# B&R Automation Studio project NAINV104C00R8L515F00
Automation Studio 4.8.4.50 SP; technology packages: Acp10Arnc0 3.18.2, mapp 1.65.1

## Configuration Inverter_Std

CPU X20CP0483, AutomationRuntime B4.82, Build 4.1.2, Safety 0.0, Vc V4.72.1

### Task classes (Cpu.sw)
```
Cyclic#1 (cycle 10000 us, tolerance 10000 us):
  DInput <- DInput.DInput.prg  // l
  DOutput <- DOutput.DOutput.prg
Cyclic#2 (cycle 20000 us, tolerance 20000 us):
  MotorBrk1 <- MotorBrk.MotorBrk.prg
  Conv <- Conv.Conv.prg
Cyclic#3 (cycle 50000 us, tolerance 50000 us):
  General <- General.General.prg
  UsrFolder <- UsrFolder.UsrFolder.prg
  Time <- Time.Time.prg
  Alarm <- Alarm.Alarm.prg
  RstErr <- RstErr.RstErr.prg
  UsrMgmt <- UsrMgmt.UsrMgmt.prg
  LibVer <- LibVer.LibVer.prg
  PneuNoSenS <- Pneu.PneuNoSenStopper.prg
  PneuNoSenC <- Pneu.PneuNoSenClamp.prg
  Pneu2SenIn <- Pneu.Pneu2SenInShutter.prg
  Pneu2SenOu <- Pneu.Pneu2SenOutShutter.prg
  Pneu2SenI1 <- Pneu.Pneu2SenInClamp1.prg
  Pneu2SenI2 <- Pneu.Pneu2SenInClamp2.prg
  Pneu2SenI3 <- Pneu.Pneu2SenInClamp3.prg
  TLBuz <- TLBuz.TLBuz.prg
  HWInfo <- HWInfo.HWInfo.prg
  ProdRcp <- ProdRcp.ProdRcp.prg
  MpProdRcp <- MpProdRcp.MpProdRcp.prg
  LCS <- LCS.LCS.prg
  LCSMngRcp <- LCS.LCSMngRcp.prg
  LCSLF <- LCS.LCSLF.prg
  Startup <- Startup.Startup.prg
  Machine <- Machine.Machine.prg
  USSMEMA <- SMEMA.USSMEMA.prg
  DSSMEMA <- SMEMA.DSSMEMA.prg
  Hermes <- Hermes.Hermes.prg
  USHermes <- Hermes.USHermes.prg
  DSHermes <- Hermes.DSHermes.prg
  RmtHermes <- Hermes.RmtHermes.prg
  LFLeader <- LF.LFLeader.prg
  LFFollower <- LF.LFFollower.prg
  Follower1 <- LF.Follower1.prg
  AWOpen <- CANOpenServo.AW.AWOpen.prg
  Ops <- Operations.Ops.prg
  OpsInvert <- Operations.OpsInvert.prg
  McParam <- McParam.McParam.prg
  NtParam <- NtParam.NtParam.prg
  UI <- UI.UI.prg
Cyclic#4 (cycle 10000 us, tolerance 10000 us):
  Simu <- Simulation.Simu.prg
  SimuInv <- Simulation.SimuInv.prg
DataObjects: Acp10sys
VcDataObjects: Visu <- UI.Visu.dob
Binaries: vccdt, vccbmp, Visu03, vcfile, arial, vctcal, arialxsr, vcmgr, vccstr, vcbclass, vccbtn, vcgclass, vcdsint, vcnet, vccline, vcshared, vccddbox, arialbd, vccnum, vcpdvnc, vcpdsw, visvc, vccslider, vccbar, vcctext, Visu01, arialbi, vcfntttf, vccovl, vccshape, vcalarm, vcpkat, Visu02, vcrt, udbdef, vccpopup, vcdsloc, vcchspot, TCData, vcpfgen, arsvcreg, Acp10map, acp10cfg, Config, iomap, User, sysconf, ashwac, ashwd, Role, asfw, arconfig, OpcUaMap, vcpfar00, segoeuib, vcctrend
Libraries: standard, astime, asstring, AsCANopen, visapi, FileIO, AsIODiag, AsMem, dvframe, AsOpcUac, sys_lib, AsTCP, runtime, AsIecCon, AsIORTI, MpRecipe, MpCom, Acp10_MC, brsystem, Acp10man, NcGlobal, Acp10par, AsFltGen, MpBase, AsUSB, vcresman, powerlnk, dataobj, asarcfg, NtUSB, NtRecipe, NtUI, NtGeneral, NtHermes
```

### Hardware
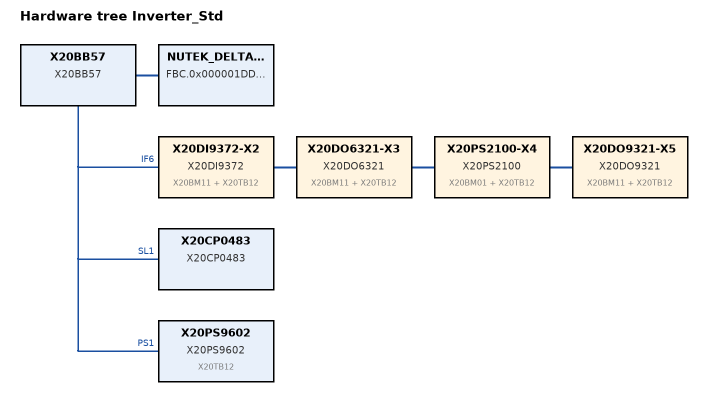
```
NUTEK_DELTA_V101 : FBC.0x000001DD.0x00000001.NUTEK_DELTA_EDS_V101 v1.0 (OrderNumber=NUTEK_DELTA_V101)  [CAN1 -> X20BB57.IF7 (NodeNumber=16)]
X20BB57 : X20BB57 v1.1.1.0
  Connector IF7:
    Baudrate = 1000000
    ActivateCanOpen = 1
    p100c_parametervalue = 1000
    p100d_parametervalue = 3
X20BM01a : X20BM01 v2.1.0.0  [X2X1 -> X20BM11c.X2X2]
X20BM11 : X20BM11 v1.0.0.1  [X2X1 -> X20BB57.IF6]
X20BM11b : X20BM11 v1.0.0.1  [X2X1 -> X20BM01a.X2X2]
X20BM11c : X20BM11 v1.0.0.1  [X2X1 -> X20BM11.X2X2]
X20CP0483 : X20CP0483 v1.2.1.0  [SL -> X20BB57.SL1]
  Connector IF2:
    ActivateDevice = 1
    Mode = Manual
    InternetAddress = 192.168.0.34
    SubnetMask = 255.255.255.0
    InaNodeNumber = 34
    Vnc1
    VncVcObjectName1 = Visu
    VncKeyMappingFile1 = VC\PS2-Keyboard.dis
    VncMaxConnections1 = 3
    VncRefreshRate1 = 100
    ActivateSnmp = 2
  ConfigurationID = NAINV104
  UserPartitionSize = 150
  EnableUsbRemoteInstall = 1
  TimerDeviceType = SWIOTIMER
  Cyclic1Duration = 10000
  Cyclic1Tolerance = 10000
  Cyclic2Duration = 20000
  Cyclic2Tolerance = 20000
  Cyclic3Duration = 50000
  Cyclic3Tolerance = 50000
  Cyclic4Duration = 10000
  Cyclic4Tolerance = 10000
  Cyclic5Duration = 150000
  Cyclic5Tolerance = 150000
  Cyclic6Duration = 500000
  Cyclic6Tolerance = 500000
  Cyclic7Duration = 1000000
  Cyclic7Tolerance = 1000000
  Cyclic8Duration = 10000
  Cyclic8Tolerance = 10000
  FileDevice1
  FileDeviceName1 = F
  FileDevicePath1 = F:
  FileDevice2
  FileDeviceName2 = User
  FileDevicePath2 = F:\User
  FileDevice3
  FileDeviceName3 = Private
  FileDevicePath3 = F:\Private
  FileDevice4
  FileDeviceName4 = CustomerUser
  FileDevicePath4 = F:\User\UserMgmt
  FileDevice5
  FileDeviceName5 = ProdRcp
  FileDevicePath5 = F:\User\ProductRecipe
  FileDevice6
  FileDeviceName6 = MagRcp
  FileDevicePath6 = F:\User\MagazineRecipe
  FileDevice7
  FileDeviceName7 = Alarm
  FileDevicePath7 = F:\User\Alarm
  FileDevice8
  FileDeviceName8 = McParam
  FileDevicePath8 = F:\User\MachineParameter
  FileDevice9
  FileDeviceName9 = NtParam
  FileDevicePath9 = F:\Private\NutekParameter
  FileDevice10
  FileDeviceName10 = LibVer
  FileDevicePath10 = F:\User\LibrariesVersion
  FileDevice11
  FileDeviceName11 = Retain
  FileDevicePath11 = F:\User\Retain
  FileDevice12
  FileDeviceName12 = Log
  FileDevicePath12 = F:\User\Log
  FileDevice13
  FileDeviceName13 = LCS
  FileDevicePath13 = F:\User\LCS
  FileDevice14
  FileDeviceName14 = MpProdRcp
  FileDevicePath14 = F:\User\ProductRecipeXml
  FileDevice15
  FileDeviceName15 = MpNtParam
  FileDevicePath15 = F:\Private\NutekParameterXml
  FtpUser1
  FtpUsername1 = NTAFTP
  FtpUserPassword1 = AX0LBkHXk5z+64iWno3s7Za7qAB1ef/xlwoQUvfPuPs=  // NTA4BH
  FtpUserSalt1 = ulQWWQjW
  FTPAccessRight1 = 0
  FTPdevice1 = ALL
  FtpUser2
  FtpUsername2 = admin
  FtpUserPassword2 = oOnwLF+CCxXL8HlJuADbdqMAHEOaZat9TyrIEGDt79E=  // admin
  FtpUserSalt2 = uTI38Rtv
  FTPAccessRight2 = 0
  FTPMSpath2 = User
  FtpUser3
  FtpUsername3 = LCS
  FtpUserPassword3 = aZ5TTuYKHpukMjerDxdtnomIopt08VfYSbHSRSZ/6LI=  // LCS
  FtpUserSalt3 = ciWQito9
  FTPAccessRight3 = 0
  FTPMSpath3 = User\LCS
  FtpUser4
  FtpUsername4 = user
  FtpUserPassword4 = iZkQD5M0oi0PmKyrQQ/mRhzQwdWVF4GSJtKjbRROesw=  // user
  FtpUserSalt4 = U6prW9t0
  FTPMSpath4 = User\ProductRecipeXml
  ActivateOpcUa = 1
  OpcUaInformationModels_PV_Version = 1
X20DI9372-X2 : X20DI9372 v1.1.0.0  [SS1 -> X20TB12a.SS; SL -> X20BM11.SL1]
X20DO6321-X3 : X20DO6321 v1.1.0.0  [SS1 -> X20TB12c.SS; SL -> X20BM11c.SL1]
X20DO9321-X5 : X20DO9321 v1.1.0.0  [SS1 -> X20TB12f.SS; SL -> X20BM11b.SL1]
X20PS2100-X4 : X20PS2100 v1.2.0.0  [SS1 -> X20TB12d.SS; SL -> X20BM01a.SL1]
X20PS9602 : X20PS9602 v1.0.2.0  [PS -> X20BB57.PS1; SS1 -> X20TB12.SS]
X20TB12 : X20TB12 v1.0.0.0
X20TB12a : X20TB12 v1.0.0.0
X20TB12c : X20TB12 v1.0.0.0
X20TB12d : X20TB12 v1.0.0.0
X20TB12f : X20TB12 v1.0.0.0
```

### IoMap.iom - X20CP0483/IoMap.iom
```iecst
VAR_CONFIG
	::DInput:a_bPhysicalDI[1] AT %IX."X20DI9372-X2".DigitalInput01;
	::DInput:a_bPhysicalDI[2] AT %IX."X20DI9372-X2".DigitalInput02;
	::DInput:a_bPhysicalDI[3] AT %IX."X20DI9372-X2".DigitalInput03;
	::DInput:a_bPhysicalDI[4] AT %IX."X20DI9372-X2".DigitalInput04;
	::DInput:a_bPhysicalDI[5] AT %IX."X20DI9372-X2".DigitalInput05;
	::DInput:a_bPhysicalDI[6] AT %IX."X20DI9372-X2".DigitalInput06;
	::DInput:a_bPhysicalDI[7] AT %IX."X20DI9372-X2".DigitalInput07;
	::DInput:a_bPhysicalDI[8] AT %IX."X20DI9372-X2".DigitalInput08;
	::DInput:a_bPhysicalDI[9] AT %IX."X20DI9372-X2".DigitalInput09;
	::DInput:a_bPhysicalDI[10] AT %IX."X20DI9372-X2".DigitalInput10;
	::DInput:a_bPhysicalDI[11] AT %IX."X20DI9372-X2".DigitalInput11;
	::DInput:a_bPhysicalDI[12] AT %IX."X20DI9372-X2".DigitalInput12;
	::AWOpen:bModuleOK AT %IX."NUTEK_DELTA_V101".ModuleOk;
	::AWOpen:tyParamOutDriver.uiCtrlword_6040 AT %QW."NUTEK_DELTA_V101".Controlword_6040;
	::AWOpen:tyParamInDriver.uiErrCode_603F AT %IW."NUTEK_DELTA_V101".ErrorCode_603F;
	::AWOpen:tyParamInDriver.uiStatword_6041 AT %IW."NUTEK_DELTA_V101".Statusword_6041;
	::AWOpen:tyParamOutDriver.siModOfOpt_6060 AT %QB."NUTEK_DELTA_V101".ModesOfOperation_6060;
	::AWOpen:tyParamInDriver.siModOfOptDisp_6061 AT %IB."NUTEK_DELTA_V101".ModesOfOperationDisplay_6061;
	::AWOpen:tyParamInDriver.diActualPos_6064 AT %ID."NUTEK_DELTA_V101".PositionActualValue_6064;
	::AWOpen:tyParamOutDriver.diTargetPos_607A AT %QD."NUTEK_DELTA_V101".TargetPosition_607A;
	::AWOpen:tyParamOutDriver.udiMoveSpd_6081 AT %QD."NUTEK_DELTA_V101".ProfileVelocity_6081;
	::AWOpen:tyParamOutDriver.siHmMethod_6098 AT %QB."NUTEK_DELTA_V101".HomingMethod_6098;
	::AWOpen:tyParamInDriver.udiDigitalInputs_60FD AT %ID."NUTEK_DELTA_V101".DigitalInputs_60FD;
	::AWOpen:tyParamOutDriver.diJogVel_60FF AT %QD."NUTEK_DELTA_V101".TargetVelocity_60FF;
	::DOutput:a_bPhysicalDO[1] AT %QX."X20DO6321-X3".DigitalOutput01;
	::DOutput:a_bPhysicalDO[2] AT %QX."X20DO6321-X3".DigitalOutput02;
	::DOutput:a_bPhysicalDO[3] AT %QX."X20DO6321-X3".DigitalOutput03;
	::DOutput:a_bPhysicalDO[4] AT %QX."X20DO6321-X3".DigitalOutput04;
	::DOutput:a_bPhysicalDO[5] AT %QX."X20DO6321-X3".DigitalOutput05;
	::DOutput:a_bPhysicalDO[6] AT %QX."X20DO6321-X3".DigitalOutput06;
	::DOutput:a_bPhysicalDO[7] AT %QX."X20DO9321".DigitalOutput01;
	::DOutput:a_bPhysicalDO[8] AT %QX."X20DO9321".DigitalOutput02;
	::DOutput:a_bPhysicalDO[9] AT %QX."X20DO9321".DigitalOutput03;
	::DOutput:a_bPhysicalDO[10] AT %QX."X20DO9321".DigitalOutput04;
	::DOutput:a_bPhysicalDO[11] AT %QX."X20DO9321".DigitalOutput05;
	::DOutput:a_bPhysicalDO[12] AT %QX."X20DO9321".DigitalOutput06;
	::DOutput:a_bPhysicalDO[13] AT %QX."X20DO9321".DigitalOutput07;
	::DOutput:a_bPhysicalDO[14] AT %QX."X20DO9321".DigitalOutput08;
	::DOutput:a_bPhysicalDO[15] AT %QX."X20DO9321".DigitalOutput09;
	::DOutput:a_bPhysicalDO[16] AT %QX."X20DO9321".DigitalOutput10;
	::DOutput:a_bPhysicalDO[17] AT %QX."X20DO9321".DigitalOutput11;
	::DOutput:a_bPhysicalDO[18] AT %QX."X20DO9321".DigitalOutput12;
	::DOutput:a_bPhysicalDO[7] AT %QX."X20DO9321-X5".DigitalOutput01;
	::DOutput:a_bPhysicalDO[8] AT %QX."X20DO9321-X5".DigitalOutput02;
	::DOutput:a_bPhysicalDO[9] AT %QX."X20DO9321-X5".DigitalOutput03;
	::DOutput:a_bPhysicalDO[10] AT %QX."X20DO9321-X5".DigitalOutput04;
	::DOutput:a_bPhysicalDO[11] AT %QX."X20DO9321-X5".DigitalOutput05;
	::DOutput:a_bPhysicalDO[12] AT %QX."X20DO9321-X5".DigitalOutput06;
	::DOutput:a_bPhysicalDO[13] AT %QX."X20DO9321-X5".DigitalOutput07;
	::DOutput:a_bPhysicalDO[14] AT %QX."X20DO9321-X5".DigitalOutput08;
	::DOutput:a_bPhysicalDO[15] AT %QX."X20DO9321-X5".DigitalOutput09;
	::DOutput:a_bPhysicalDO[16] AT %QX."X20DO9321-X5".DigitalOutput10;
	::DOutput:a_bPhysicalDO[17] AT %QX."X20DO9321-X5".DigitalOutput11;
	::DOutput:a_bPhysicalDO[18] AT %QX."X20DO9321-X5".DigitalOutput12;
END_VAR
```

## Configuration Inverter_Std_Estun

CPU X20CP0483, AutomationRuntime B4.82, Build 4.1.2, Vc V4.72.1

### Task classes (Cpu.sw)
```
Cyclic#1 (cycle 10000 us, tolerance 10000 us):
  DInput <- DInput.DInput.prg  // l
  DOutput <- DOutput.DOutput.prg
Cyclic#2 (cycle 20000 us, tolerance 20000 us):
  Conv <- Conv.Conv.prg
Cyclic#3 (cycle 50000 us, tolerance 50000 us):
  General <- General.General.prg
  UsrFolder <- UsrFolder.UsrFolder.prg
  Time <- Time.Time.prg
  Alarm <- Alarm.Alarm.prg
  RstErr <- RstErr.RstErr.prg
  UsrMgmt <- UsrMgmt.UsrMgmt.prg
  LibVer <- LibVer.LibVer.prg
  PneuNoSenS <- Pneu.PneuNoSenStopper.prg
  PneuNoSenC <- Pneu.PneuNoSenClamp.prg
  Pneu2SenIn <- Pneu.Pneu2SenInShutter.prg
  Pneu2SenOu <- Pneu.Pneu2SenOutShutter.prg
  Pneu2SenI1 <- Pneu.Pneu2SenInClamp1.prg
  Pneu2SenI2 <- Pneu.Pneu2SenInClamp2.prg
  Pneu2SenI3 <- Pneu.Pneu2SenInClamp3.prg
  TLBuz <- TLBuz.TLBuz.prg
  HWInfo <- HWInfo.HWInfo.prg
  ProdRcp <- ProdRcp.ProdRcp.prg
  MpProdRcp <- MpProdRcp.MpProdRcp.prg
  LCS <- LCS.LCS.prg
  LCSMngRcp <- LCS.LCSMngRcp.prg
  LCSLF <- LCS.LCSLF.prg
  Startup <- Startup.Startup.prg
  Machine <- Machine.Machine.prg
  MotorBrk1 <- MotorBrk.MotorBrk.prg
  USSMEMA <- SMEMA.USSMEMA.prg
  DSSMEMA <- SMEMA.DSSMEMA.prg
  Hermes <- Hermes.Hermes.prg
  USHermes <- Hermes.USHermes.prg
  DSHermes <- Hermes.DSHermes.prg
  RmtHermes <- Hermes.RmtHermes.prg
  LFLeader <- LF.LFLeader.prg
  LFFollower <- LF.LFFollower.prg
  Follower1 <- LF.Follower1.prg
  AWOpen <- CANOpenServo.AW.AWOpen.prg
  Ops <- Operations.Ops.prg
  OpsInvert <- Operations.OpsInvert.prg
  McParam <- McParam.McParam.prg
  NtParam <- NtParam.NtParam.prg
  UI <- UI.UI.prg
Cyclic#4 (cycle 10000 us, tolerance 10000 us):
  Simu <- Simulation.Simu.prg
  SimuInv <- Simulation.SimuInv.prg
DataObjects: Acp10sys
VcDataObjects: Visu <- UI.Visu.dob
Binaries: vccdt, vccbmp, Visu03, vcfile, arial, vctcal, vcmgr, vccstr, vcbclass, vccbtn, vcgclass, vcdsint, vcnet, vccline, vcshared, vccddbox, arialbd, vccnum, vcpdvnc, vcpdsw, visvc, vccslider, vccbar, vcctext, Visu01, arialbi, vcfntttf, vccovl, vccshape, vcalarm, vcpkat, Visu02, vcrt, udbdef, vccpopup, vcdsloc, vcchspot, TCData, arialxsr, vcpfgen, Acp10map, acp10cfg, Config, iomap, User, sysconf, ashwac, ashwd, Role, asfw, arconfig, vcpfar00, OpcUaMap, arsvcreg, segoeuib, vcctrend
Libraries: standard, astime, asstring, AsCANopen, visapi, FileIO, AsIODiag, AsMem, dvframe, AsOpcUac, sys_lib, AsTCP, runtime, AsIecCon, AsIORTI, MpRecipe, MpCom, Acp10_MC, brsystem, Acp10man, NcGlobal, Acp10par, AsFltGen, MpBase, AsUSB, NtMem, vcresman, powerlnk, NtBuffer, NtOvenInfo, NtRS232, NtStepper, NtFileIO, NtLogFile, NtTLBuz, NtMotion, NtPneu, NtConv, NtTCP, NtMessage, NtSMEMA, NtOPCUA, NtVersion, dataobj, asarcfg, NtLF, NtRecipe, NtUI, NtGeneral, NtHermes
```

### Hardware
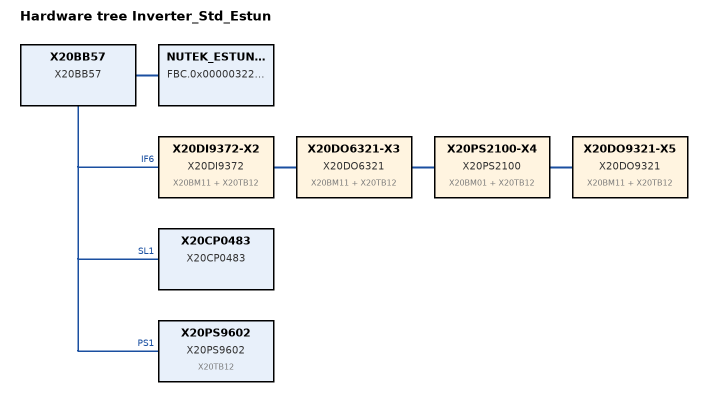
```
NUTEK_ESTUN_PronetPlus_V106 : FBC.0x00000322.0x00001000.NUTEK_ESTUN_PronetPlus_EDS_V106 v1.06.1 (OrderNumber=NUTEK_ESTUN_PronetPlus_V106)  [CAN1 -> X20BB57.IF7 (NodeNumber=16)]
X20BB57 : X20BB57 v1.1.1.0
  Connector IF7:
    Baudrate = 1000000
    ActivateCanOpen = 1
    p100c_parametervalue = 1000
    p100d_parametervalue = 3
X20BM01 : X20BM01 v2.1.0.0  [X2X1 -> X20BM11e.X2X2]
X20BM11 : X20BM11 v1.0.0.1  [X2X1 -> X20BB57.IF6]
X20BM11c : X20BM11 v1.0.0.1  [X2X1 -> X20BM01.X2X2]
X20BM11e : X20BM11 v1.0.0.1  [X2X1 -> X20BM11.X2X2]
X20CP0483 : X20CP0483 v1.2.1.0  [SL -> X20BB57.SL1]
  Connector IF2:
    ActivateDevice = 1
    Mode = Manual
    InternetAddress = 192.168.0.16
    SubnetMask = 255.255.255.0
    InaNodeNumber = 6
    Vnc1
    VncVcObjectName1 = Visu
    VncKeyMappingFile1 = VC\PS2-Keyboard.dis
    VncMaxConnections1 = 3
    VncRefreshRate1 = 100
    ActivateSnmp = 2
  ConfigurationID = NAINV104
  UserPartitionSize = 150
  EnableUsbRemoteInstall = 1
  TimerDeviceType = SWIOTIMER
  Cyclic1Duration = 10000
  Cyclic1Tolerance = 10000
  Cyclic2Duration = 20000
  Cyclic2Tolerance = 20000
  Cyclic3Duration = 50000
  Cyclic3Tolerance = 50000
  Cyclic4Duration = 10000
  Cyclic4Tolerance = 10000
  Cyclic5Duration = 150000
  Cyclic5Tolerance = 150000
  Cyclic6Duration = 500000
  Cyclic6Tolerance = 500000
  Cyclic7Duration = 1000000
  Cyclic7Tolerance = 1000000
  Cyclic8Duration = 10000
  Cyclic8Tolerance = 10000
  FileDevice1
  FileDeviceName1 = F
  FileDevicePath1 = F:
  FileDevice2
  FileDeviceName2 = User
  FileDevicePath2 = F:\User
  FileDevice3
  FileDeviceName3 = Private
  FileDevicePath3 = F:\Private
  FileDevice4
  FileDeviceName4 = CustomerUser
  FileDevicePath4 = F:\User\UserMgmt
  FileDevice5
  FileDeviceName5 = ProdRcp
  FileDevicePath5 = F:\User\ProductRecipe
  FileDevice6
  FileDeviceName6 = MagRcp
  FileDevicePath6 = F:\User\MagazineRecipe
  FileDevice7
  FileDeviceName7 = Alarm
  FileDevicePath7 = F:\User\Alarm
  FileDevice8
  FileDeviceName8 = McParam
  FileDevicePath8 = F:\User\MachineParameter
  FileDevice9
  FileDeviceName9 = NtParam
  FileDevicePath9 = F:\Private\NutekParameter
  FileDevice10
  FileDeviceName10 = LibVer
  FileDevicePath10 = F:\User\LibrariesVersion
  FileDevice11
  FileDeviceName11 = Retain
  FileDevicePath11 = F:\User\Retain
  FileDevice12
  FileDeviceName12 = Log
  FileDevicePath12 = F:\User\Log
  FileDevice13
  FileDeviceName13 = LCS
  FileDevicePath13 = F:\User\LCS
  FileDevice14
  FileDeviceName14 = MpProdRcp
  FileDevicePath14 = F:\User\ProductRecipeXml
  FileDevice15
  FileDeviceName15 = MpNtParam
  FileDevicePath15 = F:\Private\NutekParameterXml
  FtpUser1
  FtpUsername1 = NTAFTP
  FtpUserPassword1 = AX0LBkHXk5z+64iWno3s7Za7qAB1ef/xlwoQUvfPuPs=  // NTA4BH
  FtpUserSalt1 = ulQWWQjW
  FTPAccessRight1 = 0
  FTPdevice1 = ALL
  FtpUser2
  FtpUsername2 = admin
  FtpUserPassword2 = oOnwLF+CCxXL8HlJuADbdqMAHEOaZat9TyrIEGDt79E=  // admin
  FtpUserSalt2 = uTI38Rtv
  FTPAccessRight2 = 0
  FTPMSpath2 = User
  FtpUser3
  FtpUsername3 = LCS
  FtpUserPassword3 = aZ5TTuYKHpukMjerDxdtnomIopt08VfYSbHSRSZ/6LI=  // LCS
  FtpUserSalt3 = ciWQito9
  FTPAccessRight3 = 0
  FTPMSpath3 = User\LCS
  FtpUser4
  FtpUsername4 = user
  FtpUserPassword4 = JD0vxhfsk4AIsU4iEBcqNCfGv1QGBPStLuK1j+bofBk=  // user
  FtpUserSalt4 = BS0DW2Vk
  FTPMSpath4 = User\ProductRecipeXml
  ActivateOpcUa = 1
  OpcUaInformationModels_PV_Version = 1
X20DI9372-X2 : X20DI9372 v1.1.0.0  [SS1 -> X20TB12a.SS; SL -> X20BM11.SL1]
X20DO6321-X3 : X20DO6321 v1.1.0.0  [SS1 -> X20TB12e.SS; SL -> X20BM11e.SL1]
X20DO9321-X5 : X20DO9321 v1.1.0.0  [SS1 -> X20TB12c.SS; SL -> X20BM11c.SL1]
X20PS2100-X4 : X20PS2100 v1.2.0.0  [SS1 -> X20TB12f.SS; SL -> X20BM01.SL1]
X20PS9602 : X20PS9602 v1.0.2.0  [PS -> X20BB57.PS1; SS1 -> X20TB12.SS]
X20TB12 : X20TB12 v1.0.0.0
X20TB12a : X20TB12 v1.0.0.0
X20TB12c : X20TB12 v1.0.0.0
X20TB12e : X20TB12 v1.0.0.0
X20TB12f : X20TB12 v1.0.0.0
```

### IoMap.iom - X20CP0483/IoMap.iom
```iecst
VAR_CONFIG
	::DOutput:a_bPhysicalDO[7] AT %QX."X20DO9321-X5".DigitalOutput01;
	::DOutput:a_bPhysicalDO[8] AT %QX."X20DO9321-X5".DigitalOutput02;
	::DOutput:a_bPhysicalDO[9] AT %QX."X20DO9321-X5".DigitalOutput03;
	::DOutput:a_bPhysicalDO[10] AT %QX."X20DO9321-X5".DigitalOutput04;
	::DOutput:a_bPhysicalDO[11] AT %QX."X20DO9321-X5".DigitalOutput05;
	::DOutput:a_bPhysicalDO[12] AT %QX."X20DO9321-X5".DigitalOutput06;
	::DOutput:a_bPhysicalDO[13] AT %QX."X20DO9321-X5".DigitalOutput07;
	::DOutput:a_bPhysicalDO[14] AT %QX."X20DO9321-X5".DigitalOutput08;
	::DOutput:a_bPhysicalDO[15] AT %QX."X20DO9321-X5".DigitalOutput09;
	::DOutput:a_bPhysicalDO[16] AT %QX."X20DO9321-X5".DigitalOutput10;
	::DOutput:a_bPhysicalDO[17] AT %QX."X20DO9321-X5".DigitalOutput11;
	::DOutput:a_bPhysicalDO[18] AT %QX."X20DO9321-X5".DigitalOutput12;
	::DInput:a_bPhysicalDI[1] AT %IX."X20DI9372-X2".DigitalInput01;
	::DInput:a_bPhysicalDI[2] AT %IX."X20DI9372-X2".DigitalInput02;
	::DInput:a_bPhysicalDI[3] AT %IX."X20DI9372-X2".DigitalInput03;
	::DInput:a_bPhysicalDI[4] AT %IX."X20DI9372-X2".DigitalInput04;
	::DInput:a_bPhysicalDI[5] AT %IX."X20DI9372-X2".DigitalInput05;
	::DInput:a_bPhysicalDI[6] AT %IX."X20DI9372-X2".DigitalInput06;
	::DInput:a_bPhysicalDI[7] AT %IX."X20DI9372-X2".DigitalInput07;
	::DInput:a_bPhysicalDI[8] AT %IX."X20DI9372-X2".DigitalInput08;
	::DInput:a_bPhysicalDI[9] AT %IX."X20DI9372-X2".DigitalInput09;
	::DInput:a_bPhysicalDI[10] AT %IX."X20DI9372-X2".DigitalInput10;
	::DInput:a_bPhysicalDI[11] AT %IX."X20DI9372-X2".DigitalInput11;
	::DInput:a_bPhysicalDI[12] AT %IX."X20DI9372-X2".DigitalInput12;
	::DOutput:a_bPhysicalDO[1] AT %QX."X20DO6321-X3".DigitalOutput01;
	::DOutput:a_bPhysicalDO[2] AT %QX."X20DO6321-X3".DigitalOutput02;
	::DOutput:a_bPhysicalDO[3] AT %QX."X20DO6321-X3".DigitalOutput03;
	::DOutput:a_bPhysicalDO[4] AT %QX."X20DO6321-X3".DigitalOutput04;
	::DOutput:a_bPhysicalDO[5] AT %QX."X20DO6321-X3".DigitalOutput05;
	::DOutput:a_bPhysicalDO[6] AT %QX."X20DO6321-X3".DigitalOutput06;
	::AWOpen:bModuleOK AT %IX."NUTEK_ESTUN_PronetPlus_V106".ModuleOk;
	::AWOpen:tyParamInDriver.uiErrCode_603F AT %IW."NUTEK_ESTUN_PronetPlus_V106".Error_code_603F;
	::AWOpen:tyParamOutDriver.uiCtrlword_6040 AT %QW."NUTEK_ESTUN_PronetPlus_V106".Controlword_6040;
	::AWOpen:tyParamInDriver.uiStatword_6041 AT %IW."NUTEK_ESTUN_PronetPlus_V106".Statusword_6041;
	::AWOpen:tyParamOutDriver.siModOfOpt_6060 AT %QB."NUTEK_ESTUN_PronetPlus_V106".Modes_of_operation_6060;
	::AWOpen:tyParamInDriver.siModOfOptDisp_6061 AT %IB."NUTEK_ESTUN_PronetPlus_V106".Modes_of_operation_display_6061;
	::AWOpen:tyParamInDriver.diActualPos_6064 AT %ID."NUTEK_ESTUN_PronetPlus_V106".Position_actual_value_6064;
	::AWOpen:tyParamOutDriver.diTargetPos_607A AT %QD."NUTEK_ESTUN_PronetPlus_V106".Target_position_607A;
	::AWOpen:tyParamOutDriver.udiMoveSpd_6081 AT %QD."NUTEK_ESTUN_PronetPlus_V106".Profile_velocity_6081;
	::AWOpen:tyParamOutDriver.siHmMethod_6098 AT %QB."NUTEK_ESTUN_PronetPlus_V106".Homing_method_6098;
	::AWOpen:tyParamInDriver.udiDigitalInputs_60FD AT %ID."NUTEK_ESTUN_PronetPlus_V106".Digital_intputs_60FD;
	::AWOpen:tyParamOutDriver.diJogVel_60FF AT %QD."NUTEK_ESTUN_PronetPlus_V106".Target_velocity_60FF;
END_VAR
```

## Configuration Inverter_XClamp_WShutter_

### Hardware
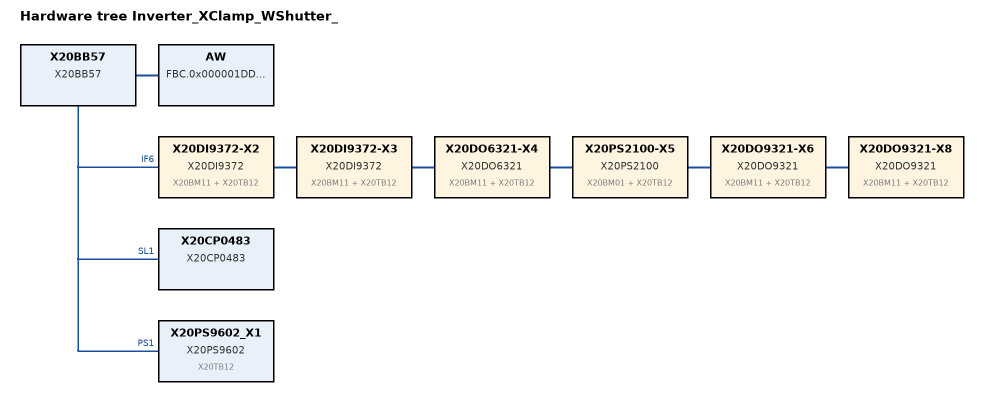
```
AW : FBC.0x000001DD.0x00000001.NUTEK_DELTA_EDS_V101 v1.0 (OrderNumber=NUTEK_DELTA_V101)  [CAN1 -> X20BB57.IF7 (NodeNumber=16)]
  Supervision = on
X20BB57 : X20BB57 v1.1.1.0
  Connector IF7:
    Baudrate = 1000000
    ActivateCanOpen = 1
    p100c_parametervalue = 1000
    p100d_parametervalue = 3
X20BM01 : X20BM01 v2.1.0.0  [X2X1 -> X20BM11a.X2X2]
X20BM11 : X20BM11 v1.0.0.1  [X2X1 -> X20BB57.IF6]
X20BM11a : X20BM11 v1.0.0.1  [X2X1 -> X20BM11e.X2X2]
X20BM11b : X20BM11 v1.0.0.1  [X2X1 -> X20BM01.X2X2]
X20BM11e : X20BM11 v1.0.0.1  [X2X1 -> X20BM11.X2X2]
X20BM11g : X20BM11 v1.0.0.1  [X2X1 -> X20BM11b.X2X2]
X20CP0483 : X20CP0483 v1.2.1.0  [SL -> X20BB57.SL1]
  Connector IF2:
    ActivateDevice = 1
    Mode = Manual
    InternetAddress = 192.168.0.30
    SubnetMask = 255.255.255.0
    InaNodeNumber = 42
    Vnc1
    VncVcObjectName1 = Visu
    VncKeyMappingFile1 = VC\PS2-Keyboard.dis
    VncMaxConnections1 = 3
    VncRefreshRate1 = 100
    ActivateSnmp = 2
  ConfigurationID = NAINV104
  UserPartitionSize = 150
  EnableUsbRemoteInstall = 1
  TimerDeviceType = SWIOTIMER
  Cyclic1Duration = 10000
  Cyclic1Tolerance = 10000
  Cyclic2Duration = 20000
  Cyclic2Tolerance = 20000
  Cyclic3Duration = 50000
  Cyclic3Tolerance = 50000
  Cyclic4Duration = 10000
  Cyclic4Tolerance = 10000
  Cyclic5Duration = 150000
  Cyclic5Tolerance = 150000
  Cyclic6Duration = 500000
  Cyclic6Tolerance = 500000
  Cyclic7Duration = 1000000
  Cyclic7Tolerance = 1000000
  Cyclic8Duration = 10000
  Cyclic8Tolerance = 10000
  FileDevice1
  FileDeviceName1 = F
  FileDevicePath1 = F:
  FileDevice2
  FileDeviceName2 = User
  FileDevicePath2 = F:\User
  FileDevice3
  FileDeviceName3 = Private
  FileDevicePath3 = F:\Private
  FileDevice4
  FileDeviceName4 = CustomerUser
  FileDevicePath4 = F:\User\UserMgmt
  FileDevice5
  FileDeviceName5 = ProdRcp
  FileDevicePath5 = F:\User\ProductRecipe
  FileDevice6
  FileDeviceName6 = MagRcp
  FileDevicePath6 = F:\User\MagazineRecipe
  FileDevice7
  FileDeviceName7 = Alarm
  FileDevicePath7 = F:\User\Alarm
  FileDevice8
  FileDeviceName8 = McParam
  FileDevicePath8 = F:\User\MachineParameter
  FileDevice9
  FileDeviceName9 = NtParam
  FileDevicePath9 = F:\Private\NutekParameter
  FileDevice10
  FileDeviceName10 = LibVer
  FileDevicePath10 = F:\User\LibrariesVersion
  FileDevice11
  FileDeviceName11 = Retain
  FileDevicePath11 = F:\User\Retain
  FileDevice12
  FileDeviceName12 = Log
  FileDevicePath12 = F:\User\Log
  FileDevice13
  FileDeviceName13 = LCS
  FileDevicePath13 = F:\User\LCS
  FileDevice14
  FileDeviceName14 = MpProdRcp
  FileDevicePath14 = F:\User\ProductRecipeXml
  FileDevice15
  FileDeviceName15 = MpNtParam
  FileDevicePath15 = F:\Private\NutekParameterXml
  FtpUser1
  FtpUsername1 = NTAFTP
  FtpUserPassword1 = AX0LBkHXk5z+64iWno3s7Za7qAB1ef/xlwoQUvfPuPs=  // NTA4BH
  FtpUserSalt1 = ulQWWQjW
  FTPAccessRight1 = 0
  FTPdevice1 = ALL
  FtpUser2
  FtpUsername2 = admin
  FtpUserPassword2 = oOnwLF+CCxXL8HlJuADbdqMAHEOaZat9TyrIEGDt79E=  // admin
  FtpUserSalt2 = uTI38Rtv
  FTPAccessRight2 = 0
  FTPMSpath2 = User
  FtpUser3
  FtpUsername3 = LCS
  FtpUserPassword3 = aZ5TTuYKHpukMjerDxdtnomIopt08VfYSbHSRSZ/6LI=  // LCS
  FtpUserSalt3 = ciWQito9
  FTPAccessRight3 = 0
  FTPMSpath3 = User\LCS
  FtpUser4
  FtpUsername4 = user
  FtpUserPassword4 = ZSNVrCTF84rK225EpwbOTF9hgjmxleDX5xeb+GcCkC0=
  FtpUserSalt4 = jV67T8tr
  FTPMSpath4 = User\ProductRecipeXml
  ActivateOpcUa = 1
  OpcUa_ConversationSecurityPolicy_EnableBasic256Rsa256 = 0
  OpcUaInformationModels_PV_Version = 1
X20DI9372-X2 : X20DI9372 v1.1.0.0  [SS1 -> X20TB12a.SS; SL -> X20BM11.SL1]
X20DI9372-X3 : X20DI9372 v1.1.0.0  [SS1 -> X20TB12g.SS; SL -> X20BM11e.SL1]
X20DO6321-X4 : X20DO6321 v1.1.0.0  [SS1 -> X20TB12b.SS; SL -> X20BM11a.SL1]
X20DO9321-X6 : X20DO9321 v1.1.0.0  [SS1 -> X20TB12c.SS; SL -> X20BM11b.SL1]
X20DO9321-X8 : X20DO9321 v1.1.0.0  [SS1 -> X20TB12i.SS; SL -> X20BM11g.SL1]
X20PS2100-X5 : X20PS2100 v1.2.0.0  [SS1 -> X20TB12f.SS; SL -> X20BM01.SL1]
X20PS9602_X1 : X20PS9602 v1.0.2.0  [PS -> X20BB57.PS1; SS1 -> X20TB12.SS]
X20TB12 : X20TB12 v1.0.0.0
X20TB12a : X20TB12 v1.0.0.0
X20TB12b : X20TB12 v1.0.0.0
X20TB12c : X20TB12 v1.0.0.0
X20TB12f : X20TB12 v1.0.0.0
X20TB12g : X20TB12 v1.0.0.0
X20TB12i : X20TB12 v1.0.0.0
```

### IoMap.iom - X20CP0483/IoMap.iom
```iecst
VAR_CONFIG
	::DInput:a_bPhysicalDI[1] AT %IX."X20DI9372-X2".DigitalInput01; (*safety relay*)
	::DInput:a_bPhysicalDI[2] AT %IX."X20DI9372-X2".DigitalInput02; (*e-stop*)
	::DInput:a_bPhysicalDI[3] AT %IX."X20DI9372-X2".DigitalInput03; (*cover swicth*)
	::DInput:a_bPhysicalDI[4] AT %IX."X20DI9372-X2".DigitalInput04; (*uba*)
	::DInput:a_bPhysicalDI[5] AT %IX."X20DI9372-X2".DigitalInput05; (*dsb*)
	::DInput:a_bPhysicalDI[6] AT %IX."X20DI9372-X2".DigitalInput06;
	::DInput:a_bPhysicalDI[7] AT %IX."X20DI9372-X2".DigitalInput07; (*inlet sen*)
	::DInput:a_bPhysicalDI[8] AT %IX."X20DI9372-X2".DigitalInput08; (*outlet sen*)
	::DInput:a_bPhysicalDI[9] AT %IX."X20DI9372-X2".DigitalInput09; (*hm inv*)
	::DInput:a_bPhysicalDI[10] AT %IX."X20DI9372-X2".DigitalInput10; (*rmt inv*)
	::DInput:a_bPhysicalDI[11] AT %IX."X20DI9372-X2".DigitalInput11; (*stp blk*)
	::DInput:a_bPhysicalDI[12] AT %IX."X20DI9372-X2".DigitalInput12; (*stp unblk*)
	::DOutput:a_bPhysicalDO[1] AT %QX."X20DO6321-X4".DigitalOutput01; (*safety relay reset*)
	::DOutput:a_bPhysicalDO[2] AT %QX."X20DO6321-X4".DigitalOutput02; (*TL G*)
	::DOutput:a_bPhysicalDO[3] AT %QX."X20DO6321-X4".DigitalOutput03; (*TL A*)
	::DOutput:a_bPhysicalDO[4] AT %QX."X20DO6321-X4".DigitalOutput04; (*TL R*)
	::DOutput:a_bPhysicalDO[5] AT %QX."X20DO6321-X4".DigitalOutput05; (*Buz*)
	::DOutput:a_bPhysicalDO[6] AT %QX."X20DO6321-X4".DigitalOutput06;
	::DOutput:a_bPhysicalDO[7] AT %QX."X20DO9321-X6".DigitalOutput01;
	::DOutput:a_bPhysicalDO[8] AT %QX."X20DO9321-X6".DigitalOutput02; (*USB*)
	::DOutput:a_bPhysicalDO[9] AT %QX."X20DO9321-X6".DigitalOutput03; (*DBA*)
	::DOutput:a_bPhysicalDO[10] AT %QX."X20DO9321-X6".DigitalOutput04;
	::DOutput:a_bPhysicalDO[11] AT %QX."X20DO9321-X6".DigitalOutput05; (*Conv Mtr CW*)
	::DOutput:a_bPhysicalDO[12] AT %QX."X20DO9321-X6".DigitalOutput06; (*Conv Mtr CWW*)
	::DOutput:a_bPhysicalDO[13] AT %QX."X20DO9321-X6".DigitalOutput07; (*Stpr ublk *)
	::DOutput:a_bPhysicalDO[14] AT %QX."X20DO9321-X6".DigitalOutput08; (*Stpr blk*)
	::DOutput:a_bPhysicalDO[15] AT %QX."X20DO9321-X6".DigitalOutput09; (*inv hm*)
	::DOutput:a_bPhysicalDO[16] AT %QX."X20DO9321-X6".DigitalOutput10; (*inv rmt*)
	::DOutput:a_bPhysicalDO[17] AT %QX."X20DO9321-X6".DigitalOutput11; (*inv brake*)
	::DOutput:a_bPhysicalDO[18] AT %QX."X20DO9321-X6".DigitalOutput12;
	::AWOpen:bModuleOK AT %IX."AW".ModuleOk;
	::AWOpen:tyParamOutDriver.uiCtrlword_6040 AT %QW."AW".Controlword_6040;
	::AWOpen:tyParamInDriver.uiStatword_6041 AT %IW."AW".Statusword_6041;
	::DInput:a_bPhysicalDI[13] AT %IX."X20DI6372".DigitalInput01;
	::DInput:a_bPhysicalDI[14] AT %IX."X20DI6372".DigitalInput02;
	::DInput:a_bPhysicalDI[15] AT %IX."X20DI6372".DigitalInput03;
	::DInput:a_bPhysicalDI[16] AT %IX."X20DI6372".DigitalInput04;
	::DInput:a_bPhysicalDI[17] AT %IX."X20DI6372".DigitalInput05;
	::DInput:a_bPhysicalDI[18] AT %IX."X20DI6372".DigitalInput06;
	::AWOpen:tyParamOutDriver.siModOfOpt_6060 AT %QB."AW".ModesOfOperation_6060;
	::AWOpen:tyParamInDriver.siModOfOptDisp_6061 AT %IB."AW".ModesOfOperationDisplay_6061;
	::AWOpen:tyParamInDriver.diActualPos_6064 AT %ID."AW".PositionActualValue_6064;
	::AWOpen:tyParamOutDriver.diTargetPos_607A AT %QD."AW".TargetPosition_607A;
	::AWOpen:tyParamOutDriver.udiMoveSpd_6081 AT %QD."AW".ProfileVelocity_6081;
	::AWOpen:tyParamOutDriver.siHmMethod_6098 AT %QB."AW".HomingMethod_6098;
	::AWOpen:tyParamInDriver.udiDigitalInputs_60FD AT %ID."AW".DigitalInputs_60FD;
	::AWOpen:tyParamOutDriver.diJogVel_60FF AT %QD."AW".TargetVelocity_60FF;
	::DInput:a_bPhysicalDI[13] AT %IX."X20DI9372-X3".DigitalInput01; (*inlet shut close reed*)
	::DInput:a_bPhysicalDI[14] AT %IX."X20DI9372-X3".DigitalInput02; (*inlet shut open reed*)
	::DInput:a_bPhysicalDI[15] AT %IX."X20DI9372-X3".DigitalInput03; (*oulet close reed*)
	::DInput:a_bPhysicalDI[16] AT %IX."X20DI9372-X3".DigitalInput04; (*outlet open reed*)
	::DInput:a_bPhysicalDI[17] AT %IX."X20DI9372-X3".DigitalInput05;
	::DInput:a_bPhysicalDI[18] AT %IX."X20DI9372-X3".DigitalInput06;
	::DInput:a_bPhysicalDI[19] AT %IX."X20DI9372-X3".DigitalInput07;
	::DInput:a_bPhysicalDI[20] AT %IX."X20DI9372-X3".DigitalInput08;
	::DInput:a_bPhysicalDI[21] AT %IX."X20DI9372-X3".DigitalInput09;
	::DInput:a_bPhysicalDI[22] AT %IX."X20DI9372-X3".DigitalInput10;
	::DInput:a_bPhysicalDI[23] AT %IX."X20DI9372-X3".DigitalInput11;
	::DInput:a_bPhysicalDI[24] AT %IX."X20DI9372-X3".DigitalInput12;
	::DOutput:a_bPhysicalDO[19] AT %QX."X20DO9321-X8".DigitalOutput01; (*inlet shut close*)
	::DOutput:a_bPhysicalDO[20] AT %QX."X20DO9321-X8".DigitalOutput02; (*inlet shut open*)
	::DOutput:a_bPhysicalDO[21] AT %QX."X20DO9321-X8".DigitalOutput03; (*outlet shut close*)
	::DOutput:a_bPhysicalDO[22] AT %QX."X20DO9321-X8".DigitalOutput04; (*outlet shut open*)
	::DOutput:a_bPhysicalDO[23] AT %QX."X20DO9321-X8".DigitalOutput05;
	::AWOpen:tyParamInDriver.uiErrCode_603F AT %IW."AW".ErrorCode_603F;
	::DOutput:a_bPhysicalDO[24] AT %QX."X20DO9321-X8".DigitalOutput06;
	::DOutput:a_bPhysicalDO[25] AT %QX."X20DO9321-X8".DigitalOutput07;
	::DOutput:a_bPhysicalDO[26] AT %QX."X20DO9321-X8".DigitalOutput08;
	::DOutput:a_bPhysicalDO[27] AT %QX."X20DO9321-X8".DigitalOutput09;
	::DOutput:a_bPhysicalDO[28] AT %QX."X20DO9321-X8".DigitalOutput10;
	::DOutput:a_bPhysicalDO[29] AT %QX."X20DO9321-X8".DigitalOutput11;
	::DOutput:a_bPhysicalDO[30] AT %QX."X20DO9321-X8".DigitalOutput12;
END_VAR
```

## Configuration Inverter_XStd_WClamp

CPU X20CP0483, AutomationRuntime B4.34, Build 4.1.2, Vc V4.33.0

### Task classes (Cpu.sw)
```
Cyclic#1 (cycle 10000 us, tolerance 10000 us):
  DInput <- DInput.DInput.prg
  DOutput <- DOutput.DOutput.prg
Cyclic#2 (cycle 20000 us, tolerance 20000 us):
  Conv <- Conv.Conv.prg
Cyclic#3 (cycle 50000 us, tolerance 50000 us):
  General <- General.General.prg
  UsrFolder <- UsrFolder.UsrFolder.prg
  Time <- Time.Time.prg
  Alarm <- Alarm.Alarm.prg
  RstErr <- RstErr.RstErr.prg
  UsrMgmt <- UsrMgmt.UsrMgmt.prg
  LibVer <- LibVer.LibVer.prg
  PneuNoSenS <- Pneu.PneuNoSenStopper.prg
  PneuNoSenC <- Pneu.PneuNoSenClamp.prg
  Pneu2SenIn <- Pneu.Pneu2SenInShutter.prg
  Pneu2SenOu <- Pneu.Pneu2SenOutShutter.prg
  Pneu2SenI1 <- Pneu.Pneu2SenInClamp1.prg
  Pneu2SenI2 <- Pneu.Pneu2SenInClamp2.prg
  Pneu2SenI3 <- Pneu.Pneu2SenInClamp3.prg
  TLBuz <- TLBuz.TLBuz.prg
  HWInfo <- HWInfo.HWInfo.prg
  LCS <- LCS.LCS.prg
  LCSMngRcp <- LCS.LCSMngRcp.prg
  Startup <- Startup.Startup.prg
  LCSLF <- LCS.LCSLF.prg
  Machine <- Machine.Machine.prg
  MotorBrk1 <- MotorBrk.MotorBrk.prg
  USSMEMA <- SMEMA.USSMEMA.prg
  DSSMEMA <- SMEMA.DSSMEMA.prg
  Hermes <- Hermes.Hermes.prg
  USHermes <- Hermes.USHermes.prg
  DSHermes <- Hermes.DSHermes.prg
  RmtHermes <- Hermes.RmtHermes.prg
  LFLeader <- LF.LFLeader.prg
  LFFollower <- LF.LFFollower.prg
  Follower1 <- LF.Follower1.prg
  AWOpen <- CANOpenServo.AW.AWOpen.prg
  Ops <- Operations.Ops.prg
  OpsInvert <- Operations.OpsInvert.prg
  McParam <- McParam.McParam.prg
  NtParam <- NtParam.NtParam.prg
  UI <- UI.UI.prg
  MpProdRcp <- MpProdRcp.MpProdRcp.prg
  ProdRcp <- ProdRcp.ProdRcp.prg
Cyclic#4 (cycle 10000 us, tolerance 10000 us):
  Simu <- Simulation.Simu.prg
  SimuInv <- Simulation.SimuInv.prg
DataObjects: Acp10sys
VcDataObjects: Visu <- UI.Visu.dob
Binaries: vccdt, vccbmp, Visu03, vcfile, arial, vctcal, arialxsr, vcmgr, vccstr, vcbclass, vccbtn, vcgclass, vcdsint, vcnet, vccline, vcshared, vccddbox, arialbd, vccnum, vcpdvnc, vcpdsw, visvc, vccslider, vccbar, vcctext, Visu01, arialbi, vcfntttf, vccovl, vccshape, vcalarm, vcpkat, Visu02, vcrt, udbdef, vccpopup, vcdsloc, vcchspot, TCData, arsvcreg, vcpfgen, arconfig, asfw, Role, ashwd, ashwac, sysconf, User, OpcUaMap, iomap, Config, acp10cfg, Acp10map, vcpfar00, segoeuib, vcctrend
Libraries: standard, astime, asstring, AsCANopen, visapi, FileIO, AsIODiag, AsMem, dvframe, AsOpcUac, sys_lib, AsTCP, runtime, AsIecCon, AsIORTI, MpRecipe, MpCom, Acp10_MC, brsystem, Acp10man, NcGlobal, Acp10par, AsFltGen, MpBase, AsRfbExt, AsUSB, vcresman, dataobj, powerlnk, asarcfg, NtRecipe, NtUI, NtGeneral, NtHermes
```

### Hardware
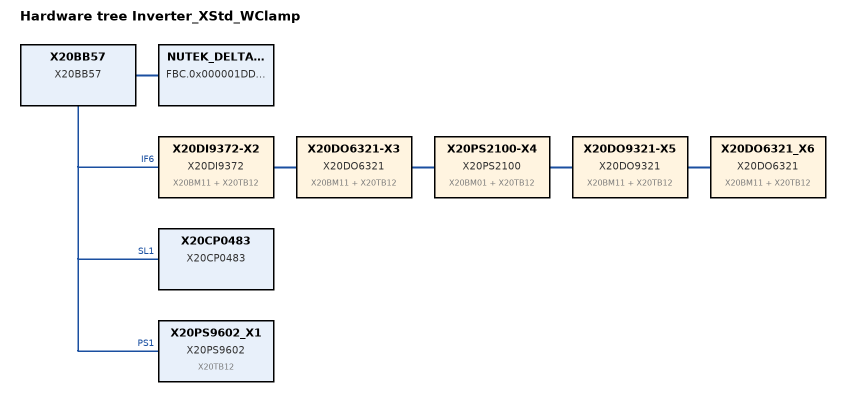
```
NUTEK_DELTA_V101 : FBC.0x000001DD.0x00000001.NUTEK_DELTA_EDS_V101 v1.0 (OrderNumber=NUTEK_DELTA_V101)  [CAN1 -> X20BB57.IF7 (NodeNumber=16)]
  Supervision = on
X20BB57 : X20BB57 v1.1.1.0
  Connector IF7:
    Baudrate = 1000000
    ActivateCanOpen = 1
    p100c_parametervalue = 1000
    p100d_parametervalue = 3
X20BM01 : X20BM01 v2.1.0.0  [X2X1 -> X20BM11a.X2X2]
X20BM11 : X20BM11 v1.0.0.1  [X2X1 -> X20BB57.IF6]
X20BM11a : X20BM11 v1.0.0.1  [X2X1 -> X20BM11.X2X2]
X20BM11b : X20BM11 v1.0.0.1  [X2X1 -> X20BM01.X2X2]
X20BM11d : X20BM11 v1.0.0.1  [X2X1 -> X20BM11b.X2X2]
X20CP0483 : X20CP0483 v1.2.1.0  [SL -> X20BB57.SL1]
  Connector IF2:
    ActivateDevice = 1
    Mode = Manual
    InternetAddress = 192.168.0.6
    SubnetMask = 255.255.255.0
    InaNodeNumber = 6
    Vnc1
    VncVcObjectName1 = Visu
    VncKeyMappingFile1 = VC\PS2-Keyboard.dis
    VncMaxConnections1 = 3
    VncRefreshRate1 = 100
  ConfigurationID = NAINV104
  UserPartitionSize = 150
  EnableUsbRemoteInstall = 1
  TimerDeviceType = SWIOTIMER
  Cyclic1Duration = 10000
  Cyclic1Tolerance = 10000
  Cyclic2Duration = 20000
  Cyclic2Tolerance = 20000
  Cyclic3Duration = 50000
  Cyclic3Tolerance = 50000
  Cyclic4Duration = 10000
  Cyclic4Tolerance = 10000
  Cyclic5Duration = 150000
  Cyclic5Tolerance = 150000
  Cyclic6Duration = 500000
  Cyclic6Tolerance = 500000
  Cyclic7Duration = 1000000
  Cyclic7Tolerance = 1000000
  Cyclic8Duration = 10000
  Cyclic8Tolerance = 10000
  FileDevice1
  FileDeviceName1 = F
  FileDevicePath1 = F:
  FileDevice2
  FileDeviceName2 = User
  FileDevicePath2 = F:\User
  FileDevice3
  FileDeviceName3 = Private
  FileDevicePath3 = F:\Private
  FileDevice4
  FileDeviceName4 = CustomerUser
  FileDevicePath4 = F:\User\UserMgmt
  FileDevice5
  FileDeviceName5 = ProdRcp
  FileDevicePath5 = F:\User\ProductRecipe
  FileDevice6
  FileDeviceName6 = MagRcp
  FileDevicePath6 = F:\User\MagazineRecipe
  FileDevice7
  FileDeviceName7 = Alarm
  FileDevicePath7 = F:\User\Alarm
  FileDevice8
  FileDeviceName8 = McParam
  FileDevicePath8 = F:\User\MachineParameter
  FileDevice9
  FileDeviceName9 = NtParam
  FileDevicePath9 = F:\Private\NutekParameter
  FileDevice10
  FileDeviceName10 = LibVer
  FileDevicePath10 = F:\User\LibrariesVersion
  FileDevice11
  FileDeviceName11 = Retain
  FileDevicePath11 = F:\User\Retain
  FileDevice12
  FileDeviceName12 = Log
  FileDevicePath12 = F:\User\Log
  FileDevice13
  FileDeviceName13 = LCS
  FileDevicePath13 = F:\User\LCS
  FileDevice14
  FileDeviceName14 = MpProdRcp
  FileDevicePath14 = F:\User\ProductRecipeXml
  FileDevice15
  FileDeviceName15 = MpNtParam
  FileDevicePath15 = F:\Private\NutekParameterXml
  FtpUser1
  FtpUsername1 = NTAFTP
  FtpUserPassword1 = AX0LBkHXk5z+64iWno3s7Za7qAB1ef/xlwoQUvfPuPs=  // NTA4BH
  FtpUserSalt1 = ulQWWQjW
  FTPAccessRight1 = 0
  FTPdevice1 = ALL
  FtpUser2
  FtpUsername2 = admin
  FtpUserPassword2 = oOnwLF+CCxXL8HlJuADbdqMAHEOaZat9TyrIEGDt79E=  // admin
  FtpUserSalt2 = uTI38Rtv
  FTPAccessRight2 = 0
  FTPMSpath2 = User
  FtpUser3
  FtpUsername3 = LCS
  FtpUserPassword3 = aZ5TTuYKHpukMjerDxdtnomIopt08VfYSbHSRSZ/6LI=  // LCS
  FtpUserSalt3 = ciWQito9
  FTPAccessRight3 = 0
  FTPMSpath3 = User\LCS
  FtpUser4
  FtpUsername4 = user
  FtpUserPassword4 = iCt/72nJS6I3I2E3ul1RgkpC9BzXhJ9PtEYmUm0QYyA=  // user
  FtpUserSalt4 = 7DfIs+80
  FTPMSpath4 = User\ProductRecipeXml
  ActivateOpcUa = 1
X20DI9372-X2 : X20DI9372 v1.1.0.0  [SS1 -> X20TB12a.SS; SL -> X20BM11.SL1]
X20DO6321-X3 : X20DO6321 v1.1.0.0  [SS1 -> X20TB12b.SS; SL -> X20BM11a.SL1]
X20DO6321_X6 : X20DO6321 v1.1.0.0  [SS1 -> X20TB12e.SS; SL -> X20BM11d.SL1]
X20DO9321-X5 : X20DO9321 v1.1.0.0  [SS1 -> X20TB12c.SS; SL -> X20BM11b.SL1]
X20PS2100-X4 : X20PS2100 v1.2.0.0  [SS1 -> X20TB12f.SS; SL -> X20BM01.SL1]
X20PS9602_X1 : X20PS9602 v1.0.2.0  [PS -> X20BB57.PS1; SS1 -> X20TB12.SS]
X20TB12 : X20TB12 v1.0.0.0
X20TB12a : X20TB12 v1.0.0.0
X20TB12b : X20TB12 v1.0.0.0
X20TB12c : X20TB12 v1.0.0.0
X20TB12e : X20TB12 v1.0.0.0
X20TB12f : X20TB12 v1.0.0.0
```

### IoMap.iom - X20CP0483/IoMap.iom
```iecst
VAR_CONFIG
	::DInput:a_bPhysicalDI[1] AT %IX."X20DI9372-X2".DigitalInput01;
	::DInput:a_bPhysicalDI[2] AT %IX."X20DI9372-X2".DigitalInput02;
	::DInput:a_bPhysicalDI[3] AT %IX."X20DI9372-X2".DigitalInput03;
	::DInput:a_bPhysicalDI[4] AT %IX."X20DI9372-X2".DigitalInput04;
	::DInput:a_bPhysicalDI[5] AT %IX."X20DI9372-X2".DigitalInput05;
	::DInput:a_bPhysicalDI[6] AT %IX."X20DI9372-X2".DigitalInput06;
	::DInput:a_bPhysicalDI[7] AT %IX."X20DI9372-X2".DigitalInput07;
	::DInput:a_bPhysicalDI[8] AT %IX."X20DI9372-X2".DigitalInput08;
	::DInput:a_bPhysicalDI[9] AT %IX."X20DI9372-X2".DigitalInput09;
	::DInput:a_bPhysicalDI[10] AT %IX."X20DI9372-X2".DigitalInput10;
	::DInput:a_bPhysicalDI[11] AT %IX."X20DI9372-X2".DigitalInput11;
	::DInput:a_bPhysicalDI[12] AT %IX."X20DI9372-X2".DigitalInput12;
	::DOutput:a_bPhysicalDO[1] AT %QX."X20DO6321-X3".DigitalOutput01;
	::DOutput:a_bPhysicalDO[2] AT %QX."X20DO6321-X3".DigitalOutput02;
	::DOutput:a_bPhysicalDO[3] AT %QX."X20DO6321-X3".DigitalOutput03;
	::DOutput:a_bPhysicalDO[4] AT %QX."X20DO6321-X3".DigitalOutput04;
	::DOutput:a_bPhysicalDO[5] AT %QX."X20DO6321-X3".DigitalOutput05;
	::DOutput:a_bPhysicalDO[6] AT %QX."X20DO6321-X3".DigitalOutput06;
	::DOutput:a_bPhysicalDO[7] AT %QX."X20DO9321-X5".DigitalOutput01;
	::DOutput:a_bPhysicalDO[8] AT %QX."X20DO9321-X5".DigitalOutput02;
	::DOutput:a_bPhysicalDO[9] AT %QX."X20DO9321-X5".DigitalOutput03;
	::DOutput:a_bPhysicalDO[10] AT %QX."X20DO9321-X5".DigitalOutput04;
	::DOutput:a_bPhysicalDO[11] AT %QX."X20DO9321-X5".DigitalOutput05;
	::DOutput:a_bPhysicalDO[12] AT %QX."X20DO9321-X5".DigitalOutput06;
	::DOutput:a_bPhysicalDO[13] AT %QX."X20DO9321-X5".DigitalOutput07;
	::DOutput:a_bPhysicalDO[14] AT %QX."X20DO9321-X5".DigitalOutput08;
	::DOutput:a_bPhysicalDO[15] AT %QX."X20DO9321-X5".DigitalOutput09;
	::DOutput:a_bPhysicalDO[16] AT %QX."X20DO9321-X5".DigitalOutput10;
	::DOutput:a_bPhysicalDO[17] AT %QX."X20DO9321-X5".DigitalOutput11;
	::DOutput:a_bPhysicalDO[18] AT %QX."X20DO9321-X5".DigitalOutput12;
	::AWOpen:bModuleOK AT %IX."NUTEK_DELTA_V101".ModuleOk;
	::AWOpen:tyParamOutDriver.uiCtrlword_6040 AT %QW."NUTEK_DELTA_V101".Controlword_6040;
	::AWOpen:tyParamInDriver.uiStatword_6041 AT %IW."NUTEK_DELTA_V101".Statusword_6041;
	::DInput:a_bPhysicalDI[13] AT %IX."X20DI6372".DigitalInput01;
	::DInput:a_bPhysicalDI[14] AT %IX."X20DI6372".DigitalInput02;
	::DInput:a_bPhysicalDI[15] AT %IX."X20DI6372".DigitalInput03;
	::DInput:a_bPhysicalDI[16] AT %IX."X20DI6372".DigitalInput04;
	::DInput:a_bPhysicalDI[17] AT %IX."X20DI6372".DigitalInput05;
	::DInput:a_bPhysicalDI[18] AT %IX."X20DI6372".DigitalInput06;
	::DOutput:a_bPhysicalDO[19] AT %QX."X20DO6321_X6".DigitalOutput01;
	::DOutput:a_bPhysicalDO[20] AT %QX."X20DO6321_X6".DigitalOutput02;
	::DOutput:a_bPhysicalDO[21] AT %QX."X20DO6321_X6".DigitalOutput03;
	::DOutput:a_bPhysicalDO[22] AT %QX."X20DO6321_X6".DigitalOutput04;
	::DOutput:a_bPhysicalDO[23] AT %QX."X20DO6321_X6".DigitalOutput05;
	::DOutput:a_bPhysicalDO[24] AT %QX."X20DO6321_X6".DigitalOutput06;
END_VAR
```

## Configuration Inverter_XStd_WOutShutter_

### Hardware
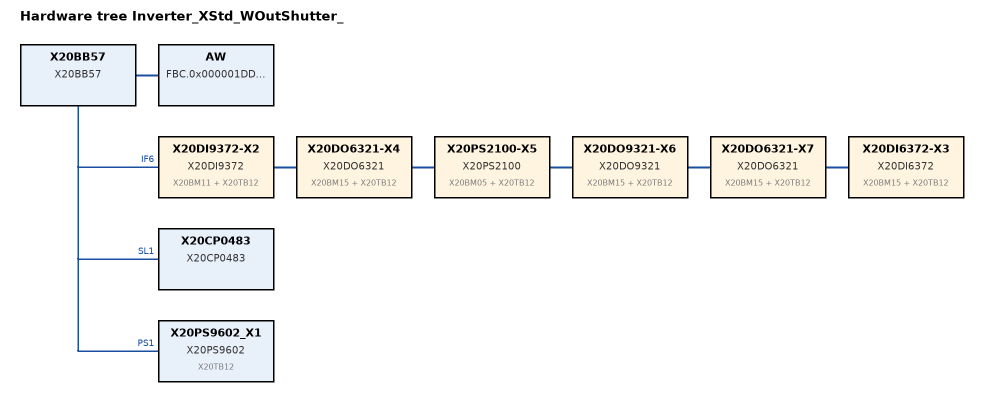
```
AW : FBC.0x000001DD.0x00000001.NUTEK_DELTA_EDS_V101 v1.0 (OrderNumber=NUTEK_DELTA_V101)  [CAN1 -> X20BB57.IF7 (NodeNumber=16)]
  Supervision = on
X20BB57 : X20BB57 v1.1.1.0
  Connector IF7:
    Baudrate = 1000000
    ActivateCanOpen = 1
    p100c_parametervalue = 1000
    p100d_parametervalue = 3
X20BM05 : X20BM05 v1.0.0.3  [X2X1 -> X20BM15b.X2X2 (NodeNumber=4)]
X20BM11 : X20BM11 v1.0.0.1  [X2X1 -> X20BB57.IF6]
X20BM15 : X20BM15 v1.0.1.0  [X2X1 -> X20BM15a.X2X2 (NodeNumber=6)]
X20BM15a : X20BM15 v1.0.1.0  [X2X1 -> X20BM05.X2X2 (NodeNumber=5)]
X20BM15b : X20BM15 v1.0.1.0  [X2X1 -> X20BM11.X2X2 (NodeNumber=3)]
X20BM15c : X20BM15 v1.0.1.0  [X2X1 -> X20BM15.X2X2 (NodeNumber=2)]
X20CP0483 : X20CP0483 v1.2.1.0  [SL -> X20BB57.SL1]
  Connector IF2:
    ActivateDevice = 1
    Mode = Manual
    InternetAddress = 192.168.0.40
    SubnetMask = 255.255.255.0
    InaNodeNumber = 40
    Vnc1
    VncVcObjectName1 = Visu
    VncKeyMappingFile1 = VC\PS2-Keyboard.dis
    VncMaxConnections1 = 3
    VncRefreshRate1 = 100
    ActivateSnmp = 2
  ConfigurationID = NAINV104
  UserPartitionSize = 150
  EnableUsbRemoteInstall = 1
  TimerDeviceType = SWIOTIMER
  Cyclic1Duration = 10000
  Cyclic1Tolerance = 10000
  Cyclic2Duration = 20000
  Cyclic2Tolerance = 20000
  Cyclic3Duration = 50000
  Cyclic3Tolerance = 50000
  Cyclic4Duration = 10000
  Cyclic4Tolerance = 10000
  Cyclic5Duration = 150000
  Cyclic5Tolerance = 150000
  Cyclic6Duration = 500000
  Cyclic6Tolerance = 500000
  Cyclic7Duration = 1000000
  Cyclic7Tolerance = 1000000
  Cyclic8Duration = 10000
  Cyclic8Tolerance = 10000
  FileDevice1
  FileDeviceName1 = F
  FileDevicePath1 = F:
  FileDevice2
  FileDeviceName2 = User
  FileDevicePath2 = F:\User
  FileDevice3
  FileDeviceName3 = Private
  FileDevicePath3 = F:\Private
  FileDevice4
  FileDeviceName4 = CustomerUser
  FileDevicePath4 = F:\User\UserMgmt
  FileDevice5
  FileDeviceName5 = ProdRcp
  FileDevicePath5 = F:\User\ProductRecipe
  FileDevice6
  FileDeviceName6 = MagRcp
  FileDevicePath6 = F:\User\MagazineRecipe
  FileDevice7
  FileDeviceName7 = Alarm
  FileDevicePath7 = F:\User\Alarm
  FileDevice8
  FileDeviceName8 = McParam
  FileDevicePath8 = F:\User\MachineParameter
  FileDevice9
  FileDeviceName9 = NtParam
  FileDevicePath9 = F:\Private\NutekParameter
  FileDevice10
  FileDeviceName10 = LibVer
  FileDevicePath10 = F:\User\LibrariesVersion
  FileDevice11
  FileDeviceName11 = Retain
  FileDevicePath11 = F:\User\Retain
  FileDevice12
  FileDeviceName12 = Log
  FileDevicePath12 = F:\User\Log
  FileDevice13
  FileDeviceName13 = LCS
  FileDevicePath13 = F:\User\LCS
  FileDevice14
  FileDeviceName14 = MpProdRcp
  FileDevicePath14 = F:\User\ProductRecipeXml
  FileDevice15
  FileDeviceName15 = MpNtParam
  FileDevicePath15 = F:\Private\NutekParameterXml
  FtpUser1
  FtpUsername1 = NTAFTP
  FtpUserPassword1 = AX0LBkHXk5z+64iWno3s7Za7qAB1ef/xlwoQUvfPuPs=  // NTA4BH
  FtpUserSalt1 = ulQWWQjW
  FTPAccessRight1 = 0
  FTPdevice1 = ALL
  FtpUser2
  FtpUsername2 = admin
  FtpUserPassword2 = oOnwLF+CCxXL8HlJuADbdqMAHEOaZat9TyrIEGDt79E=  // admin
  FtpUserSalt2 = uTI38Rtv
  FTPAccessRight2 = 0
  FTPMSpath2 = User
  FtpUser3
  FtpUsername3 = LCS
  FtpUserPassword3 = aZ5TTuYKHpukMjerDxdtnomIopt08VfYSbHSRSZ/6LI=  // LCS
  FtpUserSalt3 = ciWQito9
  FTPAccessRight3 = 0
  FTPMSpath3 = User\LCS
  FtpUser4
  FtpUsername4 = user
  FtpUserPassword4 = ZSNVrCTF84rK225EpwbOTF9hgjmxleDX5xeb+GcCkC0=
  FtpUserSalt4 = jV67T8tr
  FTPMSpath4 = User\ProductRecipeXml
  ActivateOpcUa = 1
  OpcUa_ConversationSecurityPolicy_EnableBasic256Rsa256 = 0
  OpcUaInformationModels_PV_Version = 1
X20DI6372-X3 : X20DI6372 v1.1.0.0  [SS1 -> X20TB12d.SS; SL -> X20BM15c.SL1]
X20DI9372-X2 : X20DI9372 v1.1.0.0  [SS1 -> X20TB12a.SS; SL -> X20BM11.SL1]
X20DO6321-X4 : X20DO6321 v1.1.0.0  [SS1 -> X20TB12b.SS; SL -> X20BM15b.SL1]
X20DO6321-X7 : X20DO6321 v1.1.0.0  [SS1 -> X20TB12i.SS; SL -> X20BM15.SL1]
X20DO9321-X6 : X20DO9321 v1.1.0.0  [SS1 -> X20TB12c.SS; SL -> X20BM15a.SL1]
X20PS2100-X5 : X20PS2100 v1.2.0.0  [SS1 -> X20TB12f.SS; SL -> X20BM05.SL1]
X20PS9602_X1 : X20PS9602 v1.0.2.0  [PS -> X20BB57.PS1; SS1 -> X20TB12.SS]
X20TB12 : X20TB12 v1.0.0.0
X20TB12a : X20TB12 v1.0.0.0
X20TB12b : X20TB12 v1.0.0.0
X20TB12c : X20TB12 v1.0.0.0
X20TB12d : X20TB12 v1.0.0.0
X20TB12f : X20TB12 v1.0.0.0
X20TB12i : X20TB12 v1.0.0.0
```

### IoMap.iom - X20CP0483/IoMap.iom
```iecst
VAR_CONFIG
	::DInput:a_bPhysicalDI[1] AT %IX."X20DI9372-X2".DigitalInput01;
	::DInput:a_bPhysicalDI[2] AT %IX."X20DI9372-X2".DigitalInput02;
	::DInput:a_bPhysicalDI[3] AT %IX."X20DI9372-X2".DigitalInput03;
	::DInput:a_bPhysicalDI[4] AT %IX."X20DI9372-X2".DigitalInput04;
	::DInput:a_bPhysicalDI[5] AT %IX."X20DI9372-X2".DigitalInput05;
	::DInput:a_bPhysicalDI[6] AT %IX."X20DI9372-X2".DigitalInput06;
	::DInput:a_bPhysicalDI[7] AT %IX."X20DI9372-X2".DigitalInput07;
	::DInput:a_bPhysicalDI[8] AT %IX."X20DI9372-X2".DigitalInput08;
	::DInput:a_bPhysicalDI[9] AT %IX."X20DI9372-X2".DigitalInput09;
	::DInput:a_bPhysicalDI[10] AT %IX."X20DI9372-X2".DigitalInput10;
	::DInput:a_bPhysicalDI[11] AT %IX."X20DI9372-X2".DigitalInput11;
	::DInput:a_bPhysicalDI[12] AT %IX."X20DI9372-X2".DigitalInput12;
	::DOutput:a_bPhysicalDO[1] AT %QX."X20DO6321-X4".DigitalOutput01;
	::DOutput:a_bPhysicalDO[2] AT %QX."X20DO6321-X4".DigitalOutput02;
	::DOutput:a_bPhysicalDO[3] AT %QX."X20DO6321-X4".DigitalOutput03;
	::DOutput:a_bPhysicalDO[4] AT %QX."X20DO6321-X4".DigitalOutput04;
	::DOutput:a_bPhysicalDO[5] AT %QX."X20DO6321-X4".DigitalOutput05;
	::DOutput:a_bPhysicalDO[6] AT %QX."X20DO6321-X4".DigitalOutput06;
	::DOutput:a_bPhysicalDO[7] AT %QX."X20DO9321-X6".DigitalOutput01;
	::DOutput:a_bPhysicalDO[8] AT %QX."X20DO9321-X6".DigitalOutput02;
	::DOutput:a_bPhysicalDO[9] AT %QX."X20DO9321-X6".DigitalOutput03;
	::DOutput:a_bPhysicalDO[10] AT %QX."X20DO9321-X6".DigitalOutput04;
	::DOutput:a_bPhysicalDO[11] AT %QX."X20DO9321-X6".DigitalOutput05;
	::DOutput:a_bPhysicalDO[12] AT %QX."X20DO9321-X6".DigitalOutput06;
	::DOutput:a_bPhysicalDO[13] AT %QX."X20DO9321-X6".DigitalOutput07;
	::DOutput:a_bPhysicalDO[14] AT %QX."X20DO9321-X6".DigitalOutput08;
	::DOutput:a_bPhysicalDO[15] AT %QX."X20DO9321-X6".DigitalOutput09;
	::DOutput:a_bPhysicalDO[16] AT %QX."X20DO9321-X6".DigitalOutput10;
	::DOutput:a_bPhysicalDO[17] AT %QX."X20DO9321-X6".DigitalOutput11;
	::DOutput:a_bPhysicalDO[18] AT %QX."X20DO9321-X6".DigitalOutput12;
	::AWOpen:bModuleOK AT %IX."AW".ModuleOk;
	::AWOpen:tyParamOutDriver.uiCtrlword_6040 AT %QW."AW".Controlword_6040;
	::AWOpen:tyParamInDriver.uiStatword_6041 AT %IW."AW".Statusword_6041;
	::AWOpen:tyParamOutDriver.siModOfOpt_6060 AT %QB."AW".ModesOfOperation_6060;
	::AWOpen:tyParamInDriver.siModOfOptDisp_6061 AT %IB."AW".ModesOfOperationDisplay_6061;
	::AWOpen:tyParamInDriver.diActualPos_6064 AT %ID."AW".PositionActualValue_6064;
	::AWOpen:tyParamOutDriver.diTargetPos_607A AT %QD."AW".TargetPosition_607A;
	::AWOpen:tyParamOutDriver.udiMoveSpd_6081 AT %QD."AW".ProfileVelocity_6081;
	::AWOpen:tyParamOutDriver.siHmMethod_6098 AT %QB."AW".HomingMethod_6098;
	::AWOpen:tyParamInDriver.udiDigitalInputs_60FD AT %ID."AW".DigitalInputs_60FD;
	::AWOpen:tyParamOutDriver.diJogVel_60FF AT %QD."AW".TargetVelocity_60FF;
	::DOutput:a_bPhysicalDO[19] AT %QX."X20DO6321-X7".DigitalOutput01;
	::DOutput:a_bPhysicalDO[20] AT %QX."X20DO6321-X7".DigitalOutput02;
	::DOutput:a_bPhysicalDO[21] AT %QX."X20DO6321-X7".DigitalOutput03;
	::DOutput:a_bPhysicalDO[22] AT %QX."X20DO6321-X7".DigitalOutput04;
	::DOutput:a_bPhysicalDO[23] AT %QX."X20DO6321-X7".DigitalOutput05;
	::DOutput:a_bPhysicalDO[24] AT %QX."X20DO6321-X7".DigitalOutput06;
	::AWOpen:tyParamInDriver.uiErrCode_603F AT %IW."AW".ErrorCode_603F;
	::DInput:a_bPhysicalDI[13] AT %IX."X20DI6372-X3".DigitalInput01;
	::DInput:a_bPhysicalDI[14] AT %IX."X20DI6372-X3".DigitalInput02;
	::DInput:a_bPhysicalDI[15] AT %IX."X20DI6372-X3".DigitalInput03;
	::DInput:a_bPhysicalDI[16] AT %IX."X20DI6372-X3".DigitalInput04;
	::DInput:a_bPhysicalDI[17] AT %IX."X20DI6372-X3".DigitalInput05;
	::DInput:a_bPhysicalDI[18] AT %IX."X20DI6372-X3".DigitalInput06;
END_VAR
```

## Configuration Inverter_XStd_WShutter

CPU X20CP0483, AutomationRuntime B4.82, Build 4.1.2, Vc V4.72.1

### Task classes (Cpu.sw)
```
Cyclic#1 (cycle 10000 us, tolerance 10000 us):
  DInput <- DInput.DInput.prg
  DOutput <- DOutput.DOutput.prg
Cyclic#2 (cycle 20000 us, tolerance 20000 us):
  Conv <- Conv.Conv.prg
Cyclic#3 (cycle 50000 us, tolerance 50000 us):
  General <- General.General.prg
  UsrFolder <- UsrFolder.UsrFolder.prg
  Time <- Time.Time.prg
  Alarm <- Alarm.Alarm.prg
  RstErr <- RstErr.RstErr.prg
  UsrMgmt <- UsrMgmt.UsrMgmt.prg
  LibVer <- LibVer.LibVer.prg
  PneuNoSenS <- Pneu.PneuNoSenStopper.prg
  PneuNoSenC <- Pneu.PneuNoSenClamp.prg
  Pneu2SenIn <- Pneu.Pneu2SenInShutter.prg
  Pneu2SenOu <- Pneu.Pneu2SenOutShutter.prg
  Pneu2SenI1 <- Pneu.Pneu2SenInClamp1.prg
  Pneu2SenI2 <- Pneu.Pneu2SenInClamp2.prg
  Pneu2SenI3 <- Pneu.Pneu2SenInClamp3.prg
  TLBuz <- TLBuz.TLBuz.prg
  HWInfo <- HWInfo.HWInfo.prg
  LCS <- LCS.LCS.prg
  LCSMngRcp <- LCS.LCSMngRcp.prg
  Startup <- Startup.Startup.prg
  LCSLF <- LCS.LCSLF.prg
  Machine <- Machine.Machine.prg
  MotorBrk1 <- MotorBrk.MotorBrk.prg
  USSMEMA <- SMEMA.USSMEMA.prg
  DSSMEMA <- SMEMA.DSSMEMA.prg
  Hermes <- Hermes.Hermes.prg
  USHermes <- Hermes.USHermes.prg
  DSHermes <- Hermes.DSHermes.prg
  RmtHermes <- Hermes.RmtHermes.prg
  LFLeader <- LF.LFLeader.prg
  LFFollower <- LF.LFFollower.prg
  Follower1 <- LF.Follower1.prg
  AWOpen <- CANOpenServo.AW.AWOpen.prg
  Ops <- Operations.Ops.prg
  OpsInvert <- Operations.OpsInvert.prg
  McParam <- McParam.McParam.prg
  NtParam <- NtParam.NtParam.prg
  UI <- UI.UI.prg
  MpProdRcp <- MpProdRcp.MpProdRcp.prg
  ProdRcp <- ProdRcp.ProdRcp.prg
Cyclic#4 (cycle 10000 us, tolerance 10000 us):
  Simu <- Simulation.Simu.prg
  SimuInv <- Simulation.SimuInv.prg
DataObjects: Acp10sys
VcDataObjects: Visu <- UI.Visu.dob
Binaries: vcpfgen, OpcUaMap, segoeuib, vcctrend
Libraries: standard, runtime, astime, asstring, operator, AsIecCon, AsCANopen, visapi, FileIO, AsIODiag, AsMem, dvframe, AsOpcUac, AsARCfg, sys_lib, AsTCP, AsIORTI, brsystem, AsFltGen, AsUSB, MpCom, MpBase, MpRecipe, Acp10man, Acp10par, NcGlobal, Acp10_MC, AsRfbExt, NtBuffer, NtMem, NtOvenInfo, NtRS232, NtStepper, NtFileIO, NtLogFile, NtTLBuz, NtMotion, NtPneu, NtConv, NtTCP, NtMessage, NtSMEMA, NtOPCUA, NtVersion, NtLF, NtRecipe, NtUI, NtGeneral, NtHermes
```

### Hardware
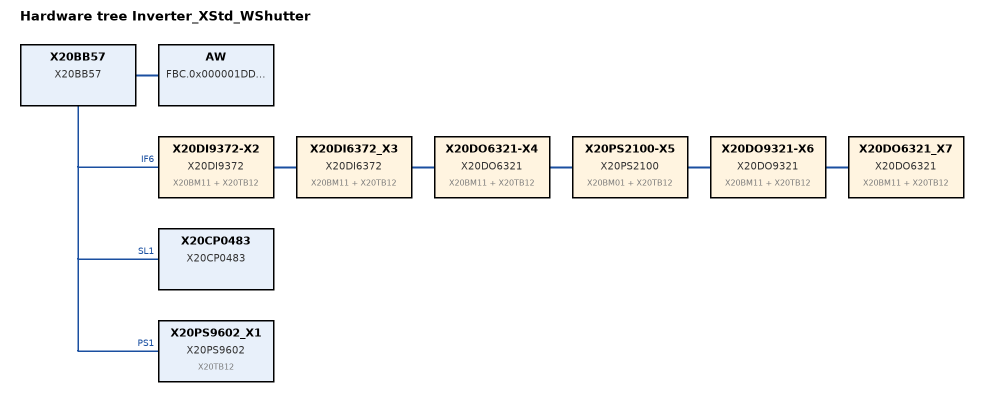
```
AW : FBC.0x000001DD.0x00000001.NUTEK_DELTA_EDS_V101 v1.0 (OrderNumber=NUTEK_DELTA_V101)  [CAN1 -> X20BB57.IF7 (NodeNumber=16)]
  Supervision = on
X20BB57 : X20BB57 v1.1.1.0
  Connector IF7:
    Baudrate = 1000000
    ActivateCanOpen = 1
    p100c_parametervalue = 1000
    p100d_parametervalue = 3
X20BM01 : X20BM01 v2.1.0.0  [X2X1 -> X20BM11a.X2X2]
X20BM11 : X20BM11 v1.0.0.1  [X2X1 -> X20BB57.IF6]
X20BM11a : X20BM11 v1.0.0.1  [X2X1 -> X20BM11c.X2X2]
X20BM11b : X20BM11 v1.0.0.1  [X2X1 -> X20BM01.X2X2]
X20BM11c : X20BM11 v1.0.0.1  [X2X1 -> X20BM11.X2X2]
X20BM11d : X20BM11 v1.0.0.1  [X2X1 -> X20BM11b.X2X2]
X20CP0483 : X20CP0483 v1.2.1.0  [SL -> X20BB57.SL1]
  Connector IF2:
    ActivateDevice = 1
    Mode = Manual
    InternetAddress = 192.168.0.14
    SubnetMask = 255.255.255.0
    InaNodeNumber = 14
    Vnc1
    VncVcObjectName1 = Visu
    VncKeyMappingFile1 = VC\PS2-Keyboard.dis
    VncMaxConnections1 = 3
    VncRefreshRate1 = 100
    ActivateSnmp = 2
  ConfigurationID = NAINV104
  UserPartitionSize = 150
  EnableUsbRemoteInstall = 1
  TimerDeviceType = SWIOTIMER
  Cyclic1Duration = 10000
  Cyclic1Tolerance = 10000
  Cyclic2Duration = 20000
  Cyclic2Tolerance = 20000
  Cyclic3Duration = 50000
  Cyclic3Tolerance = 50000
  Cyclic4Duration = 10000
  Cyclic4Tolerance = 10000
  Cyclic5Duration = 150000
  Cyclic5Tolerance = 150000
  Cyclic6Duration = 500000
  Cyclic6Tolerance = 500000
  Cyclic7Duration = 1000000
  Cyclic7Tolerance = 1000000
  Cyclic8Duration = 10000
  Cyclic8Tolerance = 10000
  FileDevice1
  FileDeviceName1 = F
  FileDevicePath1 = F:
  FileDevice2
  FileDeviceName2 = User
  FileDevicePath2 = F:\User
  FileDevice3
  FileDeviceName3 = Private
  FileDevicePath3 = F:\Private
  FileDevice4
  FileDeviceName4 = CustomerUser
  FileDevicePath4 = F:\User\UserMgmt
  FileDevice5
  FileDeviceName5 = ProdRcp
  FileDevicePath5 = F:\User\ProductRecipe
  FileDevice6
  FileDeviceName6 = MagRcp
  FileDevicePath6 = F:\User\MagazineRecipe
  FileDevice7
  FileDeviceName7 = Alarm
  FileDevicePath7 = F:\User\Alarm
  FileDevice8
  FileDeviceName8 = McParam
  FileDevicePath8 = F:\User\MachineParameter
  FileDevice9
  FileDeviceName9 = NtParam
  FileDevicePath9 = F:\Private\NutekParameter
  FileDevice10
  FileDeviceName10 = LibVer
  FileDevicePath10 = F:\User\LibrariesVersion
  FileDevice11
  FileDeviceName11 = Retain
  FileDevicePath11 = F:\User\Retain
  FileDevice12
  FileDeviceName12 = Log
  FileDevicePath12 = F:\User\Log
  FileDevice13
  FileDeviceName13 = LCS
  FileDevicePath13 = F:\User\LCS
  FileDevice14
  FileDeviceName14 = MpProdRcp
  FileDevicePath14 = F:\User\ProductRecipeXml
  FileDevice15
  FileDeviceName15 = MpNtParam
  FileDevicePath15 = F:\Private\NutekParameterXml
  FtpUser1
  FtpUsername1 = NTAFTP
  FtpUserPassword1 = AX0LBkHXk5z+64iWno3s7Za7qAB1ef/xlwoQUvfPuPs=  // NTA4BH
  FtpUserSalt1 = ulQWWQjW
  FTPAccessRight1 = 0
  FTPdevice1 = ALL
  FtpUser2
  FtpUsername2 = admin
  FtpUserPassword2 = oOnwLF+CCxXL8HlJuADbdqMAHEOaZat9TyrIEGDt79E=  // admin
  FtpUserSalt2 = uTI38Rtv
  FTPAccessRight2 = 0
  FTPMSpath2 = User
  FtpUser3
  FtpUsername3 = LCS
  FtpUserPassword3 = aZ5TTuYKHpukMjerDxdtnomIopt08VfYSbHSRSZ/6LI=  // LCS
  FtpUserSalt3 = ciWQito9
  FTPAccessRight3 = 0
  FTPMSpath3 = User\LCS
  FtpUser4
  FtpUsername4 = user
  FtpUserPassword4 = ZSNVrCTF84rK225EpwbOTF9hgjmxleDX5xeb+GcCkC0=
  FtpUserSalt4 = jV67T8tr
  FTPMSpath4 = User\ProductRecipeXml
  ActivateOpcUa = 1
  OpcUa_ConversationSecurityPolicy_EnableBasic256Rsa256 = 0
  OpcUaInformationModels_PV_Version = 1
X20DI6372_X3 : X20DI6372 v1.1.0.0  [SS1 -> X20TB12d.SS; SL -> X20BM11c.SL1]
X20DI9372-X2 : X20DI9372 v1.1.0.0  [SS1 -> X20TB12a.SS; SL -> X20BM11.SL1]
X20DO6321-X4 : X20DO6321 v1.1.0.0  [SS1 -> X20TB12b.SS; SL -> X20BM11a.SL1]
X20DO6321_X7 : X20DO6321 v1.1.0.0  [SS1 -> X20TB12e.SS; SL -> X20BM11d.SL1]
X20DO9321-X6 : X20DO9321 v1.1.0.0  [SS1 -> X20TB12c.SS; SL -> X20BM11b.SL1]
X20PS2100-X5 : X20PS2100 v1.2.0.0  [SS1 -> X20TB12f.SS; SL -> X20BM01.SL1]
X20PS9602_X1 : X20PS9602 v1.0.2.0  [PS -> X20BB57.PS1; SS1 -> X20TB12.SS]
X20TB12 : X20TB12 v1.0.0.0
X20TB12a : X20TB12 v1.0.0.0
X20TB12b : X20TB12 v1.0.0.0
X20TB12c : X20TB12 v1.0.0.0
X20TB12d : X20TB12 v1.0.0.0
X20TB12e : X20TB12 v1.0.0.0
X20TB12f : X20TB12 v1.0.0.0
```

### IoMap.iom - X20CP0483/IoMap.iom
```iecst
VAR_CONFIG
	::DInput:a_bPhysicalDI[1] AT %IX."X20DI9372-X2".DigitalInput01;
	::DInput:a_bPhysicalDI[2] AT %IX."X20DI9372-X2".DigitalInput02;
	::DInput:a_bPhysicalDI[3] AT %IX."X20DI9372-X2".DigitalInput03;
	::DInput:a_bPhysicalDI[4] AT %IX."X20DI9372-X2".DigitalInput04;
	::DInput:a_bPhysicalDI[5] AT %IX."X20DI9372-X2".DigitalInput05;
	::DInput:a_bPhysicalDI[6] AT %IX."X20DI9372-X2".DigitalInput06;
	::DInput:a_bPhysicalDI[7] AT %IX."X20DI9372-X2".DigitalInput07;
	::DInput:a_bPhysicalDI[8] AT %IX."X20DI9372-X2".DigitalInput08;
	::DInput:a_bPhysicalDI[9] AT %IX."X20DI9372-X2".DigitalInput09;
	::DInput:a_bPhysicalDI[10] AT %IX."X20DI9372-X2".DigitalInput10;
	::DInput:a_bPhysicalDI[11] AT %IX."X20DI9372-X2".DigitalInput11;
	::DInput:a_bPhysicalDI[12] AT %IX."X20DI9372-X2".DigitalInput12;
	::DOutput:a_bPhysicalDO[1] AT %QX."X20DO6321-X4".DigitalOutput01;
	::DOutput:a_bPhysicalDO[2] AT %QX."X20DO6321-X4".DigitalOutput02;
	::DOutput:a_bPhysicalDO[3] AT %QX."X20DO6321-X4".DigitalOutput03;
	::DOutput:a_bPhysicalDO[4] AT %QX."X20DO6321-X4".DigitalOutput04;
	::DOutput:a_bPhysicalDO[5] AT %QX."X20DO6321-X4".DigitalOutput05;
	::DOutput:a_bPhysicalDO[6] AT %QX."X20DO6321-X4".DigitalOutput06;
	::DOutput:a_bPhysicalDO[7] AT %QX."X20DO9321-X6".DigitalOutput01;
	::DOutput:a_bPhysicalDO[8] AT %QX."X20DO9321-X6".DigitalOutput02;
	::DOutput:a_bPhysicalDO[9] AT %QX."X20DO9321-X6".DigitalOutput03;
	::DOutput:a_bPhysicalDO[10] AT %QX."X20DO9321-X6".DigitalOutput04;
	::DOutput:a_bPhysicalDO[11] AT %QX."X20DO9321-X6".DigitalOutput05;
	::DOutput:a_bPhysicalDO[12] AT %QX."X20DO9321-X6".DigitalOutput06;
	::DOutput:a_bPhysicalDO[13] AT %QX."X20DO9321-X6".DigitalOutput07;
	::DOutput:a_bPhysicalDO[14] AT %QX."X20DO9321-X6".DigitalOutput08;
	::DOutput:a_bPhysicalDO[15] AT %QX."X20DO9321-X6".DigitalOutput09;
	::DOutput:a_bPhysicalDO[16] AT %QX."X20DO9321-X6".DigitalOutput10;
	::DOutput:a_bPhysicalDO[17] AT %QX."X20DO9321-X6".DigitalOutput11;
	::DOutput:a_bPhysicalDO[18] AT %QX."X20DO9321-X6".DigitalOutput12;
	::AWOpen:bModuleOK AT %IX."AW".ModuleOk;
	::AWOpen:tyParamOutDriver.uiCtrlword_6040 AT %QW."AW".Controlword_6040;
	::AWOpen:tyParamInDriver.uiStatword_6041 AT %IW."AW".Statusword_6041;
	::DInput:a_bPhysicalDI[13] AT %IX."X20DI6372".DigitalInput01;
	::DInput:a_bPhysicalDI[14] AT %IX."X20DI6372".DigitalInput02;
	::DInput:a_bPhysicalDI[15] AT %IX."X20DI6372".DigitalInput03;
	::DInput:a_bPhysicalDI[16] AT %IX."X20DI6372".DigitalInput04;
	::DInput:a_bPhysicalDI[17] AT %IX."X20DI6372".DigitalInput05;
	::DInput:a_bPhysicalDI[18] AT %IX."X20DI6372".DigitalInput06;
	::DOutput:a_bPhysicalDO[19] AT %QX."X20DO6321_X7".DigitalOutput01;
	::DOutput:a_bPhysicalDO[20] AT %QX."X20DO6321_X7".DigitalOutput02;
	::DOutput:a_bPhysicalDO[21] AT %QX."X20DO6321_X7".DigitalOutput03;
	::DOutput:a_bPhysicalDO[22] AT %QX."X20DO6321_X7".DigitalOutput04;
	::DOutput:a_bPhysicalDO[23] AT %QX."X20DO6321_X7".DigitalOutput05;
	::DOutput:a_bPhysicalDO[24] AT %QX."X20DO6321_X7".DigitalOutput06;
	::DInput:a_bPhysicalDI[13]  AT %IX."X20DI6372_X3".DigitalInput01;
	::DInput:a_bPhysicalDI[14] AT %IX."X20DI6372_X3".DigitalInput02;
	::DInput:a_bPhysicalDI[15] AT %IX."X20DI6372_X3".DigitalInput03;
	::DInput:a_bPhysicalDI[16] AT %IX."X20DI6372_X3".DigitalInput04;
	::DInput:a_bPhysicalDI[17] AT %IX."X20DI6372_X3".DigitalInput05;
	::DInput:a_bPhysicalDI[18] AT %IX."X20DI6372_X3".DigitalInput06;
	::AWOpen:tyParamOutDriver.siModOfOpt_6060 AT %QB."AW".ModesOfOperation_6060;
	::AWOpen:tyParamInDriver.siModOfOptDisp_6061 AT %IB."AW".ModesOfOperationDisplay_6061;
	::AWOpen:tyParamInDriver.diActualPos_6064 AT %ID."AW".PositionActualValue_6064;
	::AWOpen:tyParamOutDriver.diTargetPos_607A AT %QD."AW".TargetPosition_607A;
	::AWOpen:tyParamOutDriver.udiMoveSpd_6081 AT %QD."AW".ProfileVelocity_6081;
	::AWOpen:tyParamOutDriver.siHmMethod_6098 AT %QB."AW".HomingMethod_6098;
	::AWOpen:tyParamInDriver.udiDigitalInputs_60FD AT %ID."AW".DigitalInputs_60FD;
	::AWOpen:tyParamOutDriver.diJogVel_60FF AT %QD."AW".TargetVelocity_60FF;
END_VAR
```

## Configuration Inverter_XStd_WShutter_SafetySig

CPU X20CP0483, AutomationRuntime B4.82, Build 4.1.2, Safety 0.0, Vc V4.72.1

### Hardware
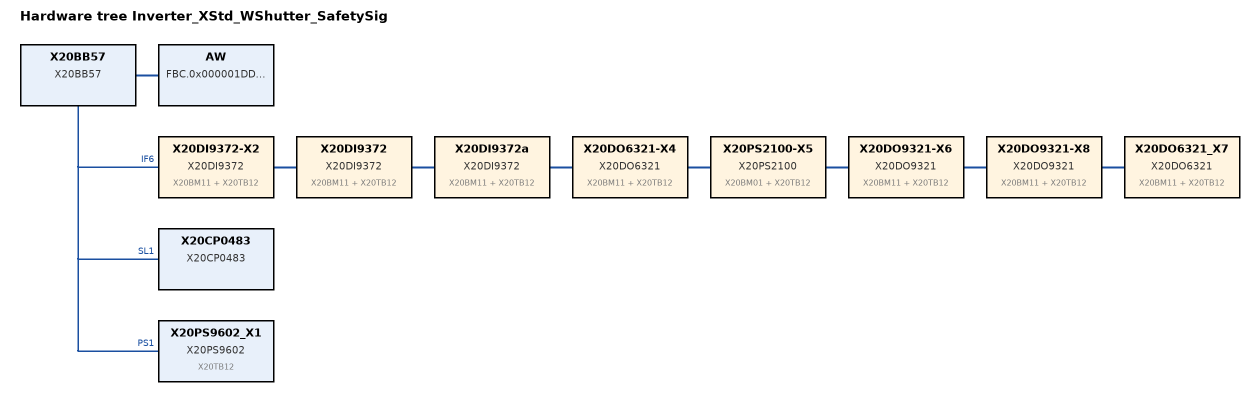
```
AW : FBC.0x000001DD.0x00000001.NUTEK_DELTA_EDS_V101 v1.0 (OrderNumber=NUTEK_DELTA_V101)  [CAN1 -> X20BB57.IF7 (NodeNumber=16)]
  Supervision = on
X20BB57 : X20BB57 v1.1.1.0
  Connector IF7:
    Baudrate = 1000000
    ActivateCanOpen = 1
    p100c_parametervalue = 1000
    p100d_parametervalue = 3
X20BM01 : X20BM01 v2.1.0.0  [X2X1 -> X20BM11a.X2X2]
X20BM11 : X20BM11 v1.0.0.1  [X2X1 -> X20BB57.IF6]
X20BM11a : X20BM11 v1.0.0.1  [X2X1 -> X20BM11f.X2X2]
X20BM11b : X20BM11 v1.0.0.1  [X2X1 -> X20BM01.X2X2]
X20BM11d : X20BM11 v1.0.0.1  [X2X1 -> X20BM11g.X2X2]
X20BM11e : X20BM11 v1.0.0.1  [X2X1 -> X20BM11.X2X2]
X20BM11f : X20BM11 v1.0.0.1  [X2X1 -> X20BM11e.X2X2]
X20BM11g : X20BM11 v1.0.0.1  [X2X1 -> X20BM11b.X2X2]
X20CP0483 : X20CP0483 v1.2.1.0  [SL -> X20BB57.SL1]
  Connector IF2:
    ActivateDevice = 1
    Mode = Manual
    InternetAddress = 192.168.0.34
    SubnetMask = 255.255.255.0
    InaNodeNumber = 42
    Vnc1
    VncVcObjectName1 = Visu
    VncKeyMappingFile1 = VC\PS2-Keyboard.dis
    VncMaxConnections1 = 3
    VncRefreshRate1 = 100
    ActivateSnmp = 2
  ConfigurationID = NAINV104
  UserPartitionSize = 150
  EnableUsbRemoteInstall = 1
  TimerDeviceType = SWIOTIMER
  Cyclic1Duration = 10000
  Cyclic1Tolerance = 10000
  Cyclic2Duration = 20000
  Cyclic2Tolerance = 20000
  Cyclic3Duration = 50000
  Cyclic3Tolerance = 50000
  Cyclic4Duration = 10000
  Cyclic4Tolerance = 10000
  Cyclic5Duration = 150000
  Cyclic5Tolerance = 150000
  Cyclic6Duration = 500000
  Cyclic6Tolerance = 500000
  Cyclic7Duration = 1000000
  Cyclic7Tolerance = 1000000
  Cyclic8Duration = 10000
  Cyclic8Tolerance = 10000
  FileDevice1
  FileDeviceName1 = F
  FileDevicePath1 = F:
  FileDevice2
  FileDeviceName2 = User
  FileDevicePath2 = F:\User
  FileDevice3
  FileDeviceName3 = Private
  FileDevicePath3 = F:\Private
  FileDevice4
  FileDeviceName4 = CustomerUser
  FileDevicePath4 = F:\User\UserMgmt
  FileDevice5
  FileDeviceName5 = ProdRcp
  FileDevicePath5 = F:\User\ProductRecipe
  FileDevice6
  FileDeviceName6 = MagRcp
  FileDevicePath6 = F:\User\MagazineRecipe
  FileDevice7
  FileDeviceName7 = Alarm
  FileDevicePath7 = F:\User\Alarm
  FileDevice8
  FileDeviceName8 = McParam
  FileDevicePath8 = F:\User\MachineParameter
  FileDevice9
  FileDeviceName9 = NtParam
  FileDevicePath9 = F:\Private\NutekParameter
  FileDevice10
  FileDeviceName10 = LibVer
  FileDevicePath10 = F:\User\LibrariesVersion
  FileDevice11
  FileDeviceName11 = Retain
  FileDevicePath11 = F:\User\Retain
  FileDevice12
  FileDeviceName12 = Log
  FileDevicePath12 = F:\User\Log
  FileDevice13
  FileDeviceName13 = LCS
  FileDevicePath13 = F:\User\LCS
  FileDevice14
  FileDeviceName14 = MpProdRcp
  FileDevicePath14 = F:\User\ProductRecipeXml
  FileDevice15
  FileDeviceName15 = MpNtParam
  FileDevicePath15 = F:\Private\NutekParameterXml
  FtpUser1
  FtpUsername1 = NTAFTP
  FtpUserPassword1 = AX0LBkHXk5z+64iWno3s7Za7qAB1ef/xlwoQUvfPuPs=  // NTA4BH
  FtpUserSalt1 = ulQWWQjW
  FTPAccessRight1 = 0
  FTPdevice1 = ALL
  FtpUser2
  FtpUsername2 = admin
  FtpUserPassword2 = oOnwLF+CCxXL8HlJuADbdqMAHEOaZat9TyrIEGDt79E=  // admin
  FtpUserSalt2 = uTI38Rtv
  FTPAccessRight2 = 0
  FTPMSpath2 = User
  FtpUser3
  FtpUsername3 = LCS
  FtpUserPassword3 = aZ5TTuYKHpukMjerDxdtnomIopt08VfYSbHSRSZ/6LI=  // LCS
  FtpUserSalt3 = ciWQito9
  FTPAccessRight3 = 0
  FTPMSpath3 = User\LCS
  FtpUser4
  FtpUsername4 = user
  FtpUserPassword4 = ZSNVrCTF84rK225EpwbOTF9hgjmxleDX5xeb+GcCkC0=
  FtpUserSalt4 = jV67T8tr
  FTPMSpath4 = User\ProductRecipeXml
  ActivateOpcUa = 1
  OpcUa_ConversationSecurityPolicy_EnableBasic256Rsa256 = 0
  OpcUaInformationModels_PV_Version = 1
X20DI9372 : X20DI9372 v1.1.0.0  [SS1 -> X20TB12g.SS; SL -> X20BM11e.SL1]
X20DI9372-X2 : X20DI9372 v1.1.0.0  [SS1 -> X20TB12a.SS; SL -> X20BM11.SL1]
X20DI9372a : X20DI9372 v1.1.0.0  [SS1 -> X20TB12h.SS; SL -> X20BM11f.SL1]
X20DO6321-X4 : X20DO6321 v1.1.0.0  [SS1 -> X20TB12b.SS; SL -> X20BM11a.SL1]
X20DO6321_X7 : X20DO6321 v1.1.0.0  [SS1 -> X20TB12e.SS; SL -> X20BM11d.SL1]
X20DO9321-X6 : X20DO9321 v1.1.0.0  [SS1 -> X20TB12c.SS; SL -> X20BM11b.SL1]
X20DO9321-X8 : X20DO9321 v1.1.0.0  [SS1 -> X20TB12i.SS; SL -> X20BM11g.SL1]
X20PS2100-X5 : X20PS2100 v1.2.0.0  [SS1 -> X20TB12f.SS; SL -> X20BM01.SL1]
X20PS9602_X1 : X20PS9602 v1.0.2.0  [PS -> X20BB57.PS1; SS1 -> X20TB12.SS]
X20TB12 : X20TB12 v1.0.0.0
X20TB12a : X20TB12 v1.0.0.0
X20TB12b : X20TB12 v1.0.0.0
X20TB12c : X20TB12 v1.0.0.0
X20TB12e : X20TB12 v1.0.0.0
X20TB12f : X20TB12 v1.0.0.0
X20TB12g : X20TB12 v1.0.0.0
X20TB12h : X20TB12 v1.0.0.0
X20TB12i : X20TB12 v1.0.0.0
```

### IoMap.iom - X20CP0483/IoMap.iom
```iecst
VAR_CONFIG
	::DInput:a_bPhysicalDI[1] AT %IX."X20DI9372-X2".DigitalInput01;
	::DInput:a_bPhysicalDI[2] AT %IX."X20DI9372-X2".DigitalInput02;
	::DInput:a_bPhysicalDI[3] AT %IX."X20DI9372-X2".DigitalInput03;
	::DInput:a_bPhysicalDI[4] AT %IX."X20DI9372-X2".DigitalInput04;
	::DInput:a_bPhysicalDI[5] AT %IX."X20DI9372-X2".DigitalInput05;
	::DInput:a_bPhysicalDI[6] AT %IX."X20DI9372-X2".DigitalInput06;
	::DInput:a_bPhysicalDI[7] AT %IX."X20DI9372-X2".DigitalInput07;
	::DInput:a_bPhysicalDI[8] AT %IX."X20DI9372-X2".DigitalInput08;
	::DInput:a_bPhysicalDI[9] AT %IX."X20DI9372-X2".DigitalInput09;
	::DInput:a_bPhysicalDI[10] AT %IX."X20DI9372-X2".DigitalInput10;
	::DInput:a_bPhysicalDI[11] AT %IX."X20DI9372-X2".DigitalInput11;
	::DInput:a_bPhysicalDI[12] AT %IX."X20DI9372-X2".DigitalInput12;
	::DOutput:a_bPhysicalDO[1] AT %QX."X20DO6321-X4".DigitalOutput01;
	::DOutput:a_bPhysicalDO[2] AT %QX."X20DO6321-X4".DigitalOutput02;
	::DOutput:a_bPhysicalDO[3] AT %QX."X20DO6321-X4".DigitalOutput03;
	::DOutput:a_bPhysicalDO[4] AT %QX."X20DO6321-X4".DigitalOutput04;
	::DOutput:a_bPhysicalDO[5] AT %QX."X20DO6321-X4".DigitalOutput05;
	::DOutput:a_bPhysicalDO[6] AT %QX."X20DO6321-X4".DigitalOutput06;
	::DOutput:a_bPhysicalDO[7] AT %QX."X20DO9321-X6".DigitalOutput01;
	::DOutput:a_bPhysicalDO[8] AT %QX."X20DO9321-X6".DigitalOutput02;
	::DOutput:a_bPhysicalDO[9] AT %QX."X20DO9321-X6".DigitalOutput03;
	::DOutput:a_bPhysicalDO[10] AT %QX."X20DO9321-X6".DigitalOutput04;
	::DOutput:a_bPhysicalDO[11] AT %QX."X20DO9321-X6".DigitalOutput05;
	::DOutput:a_bPhysicalDO[12] AT %QX."X20DO9321-X6".DigitalOutput06;
	::DOutput:a_bPhysicalDO[13] AT %QX."X20DO9321-X6".DigitalOutput07;
	::DOutput:a_bPhysicalDO[14] AT %QX."X20DO9321-X6".DigitalOutput08;
	::DOutput:a_bPhysicalDO[15] AT %QX."X20DO9321-X6".DigitalOutput09;
	::DOutput:a_bPhysicalDO[16] AT %QX."X20DO9321-X6".DigitalOutput10;
	::DOutput:a_bPhysicalDO[17] AT %QX."X20DO9321-X6".DigitalOutput11;
	::DOutput:a_bPhysicalDO[18] AT %QX."X20DO9321-X6".DigitalOutput12;
	::AWOpen:bModuleOK AT %IX."AW".ModuleOk;
	::AWOpen:tyParamOutDriver.uiCtrlword_6040 AT %QW."AW".Controlword_6040;
	::AWOpen:tyParamInDriver.uiStatword_6041 AT %IW."AW".Statusword_6041;
	::DInput:a_bPhysicalDI[13] AT %IX."X20DI6372".DigitalInput01;
	::DInput:a_bPhysicalDI[14] AT %IX."X20DI6372".DigitalInput02;
	::DInput:a_bPhysicalDI[15] AT %IX."X20DI6372".DigitalInput03;
	::DInput:a_bPhysicalDI[16] AT %IX."X20DI6372".DigitalInput04;
	::DInput:a_bPhysicalDI[17] AT %IX."X20DI6372".DigitalInput05;
	::DInput:a_bPhysicalDI[18] AT %IX."X20DI6372".DigitalInput06;
	::DOutput:a_bPhysicalDO[31] AT %QX."X20DO6321_X7".DigitalOutput01;
	::DOutput:a_bPhysicalDO[32] AT %QX."X20DO6321_X7".DigitalOutput02;
	::DOutput:a_bPhysicalDO[33] AT %QX."X20DO6321_X7".DigitalOutput03;
	::DOutput:a_bPhysicalDO[34] AT %QX."X20DO6321_X7".DigitalOutput04;
	::DOutput:a_bPhysicalDO[35] AT %QX."X20DO6321_X7".DigitalOutput05;
	::DOutput:a_bPhysicalDO[36] AT %QX."X20DO6321_X7".DigitalOutput06;
	::AWOpen:tyParamOutDriver.siModOfOpt_6060 AT %QB."AW".ModesOfOperation_6060;
	::AWOpen:tyParamInDriver.siModOfOptDisp_6061 AT %IB."AW".ModesOfOperationDisplay_6061;
	::AWOpen:tyParamInDriver.diActualPos_6064 AT %ID."AW".PositionActualValue_6064;
	::AWOpen:tyParamOutDriver.diTargetPos_607A AT %QD."AW".TargetPosition_607A;
	::AWOpen:tyParamOutDriver.udiMoveSpd_6081 AT %QD."AW".ProfileVelocity_6081;
	::AWOpen:tyParamOutDriver.siHmMethod_6098 AT %QB."AW".HomingMethod_6098;
	::AWOpen:tyParamInDriver.udiDigitalInputs_60FD AT %ID."AW".DigitalInputs_60FD;
	::AWOpen:tyParamOutDriver.diJogVel_60FF AT %QD."AW".TargetVelocity_60FF;
	::DInput:a_bPhysicalDI[13] AT %IX."X20DI9372".DigitalInput01;
	::DInput:a_bPhysicalDI[14] AT %IX."X20DI9372".DigitalInput02;
	::DInput:a_bPhysicalDI[15] AT %IX."X20DI9372".DigitalInput03;
	::DInput:a_bPhysicalDI[16] AT %IX."X20DI9372".DigitalInput04;
	::DInput:a_bPhysicalDI[17] AT %IX."X20DI9372".DigitalInput05;
	::DInput:a_bPhysicalDI[18] AT %IX."X20DI9372".DigitalInput06;
	::DInput:a_bPhysicalDI[19] AT %IX."X20DI9372".DigitalInput07;
	::DInput:a_bPhysicalDI[20] AT %IX."X20DI9372".DigitalInput08;
	::DInput:a_bPhysicalDI[21] AT %IX."X20DI9372".DigitalInput09;
	::DInput:a_bPhysicalDI[22] AT %IX."X20DI9372".DigitalInput10;
	::DInput:a_bPhysicalDI[23] AT %IX."X20DI9372".DigitalInput11;
	::DInput:a_bPhysicalDI[24] AT %IX."X20DI9372".DigitalInput12;
	::DInput:a_bPhysicalDI[25] AT %IX."X20DI9372a".DigitalInput01;
	::DInput:a_bPhysicalDI[26] AT %IX."X20DI9372a".DigitalInput02;
	::DInput:a_bPhysicalDI[27] AT %IX."X20DI9372a".DigitalInput03;
	::DInput:a_bPhysicalDI[28] AT %IX."X20DI9372a".DigitalInput04;
	::DInput:a_bPhysicalDI[29] AT %IX."X20DI9372a".DigitalInput05;
	::DInput:a_bPhysicalDI[30] AT %IX."X20DI9372a".DigitalInput06;
	::DInput:a_bPhysicalDI[31] AT %IX."X20DI9372a".DigitalInput07;
	::DInput:a_bPhysicalDI[32] AT %IX."X20DI9372a".DigitalInput08;
	::DInput:a_bPhysicalDI[33] AT %IX."X20DI9372a".DigitalInput09;
	::DInput:a_bPhysicalDI[34] AT %IX."X20DI9372a".DigitalInput10;
	::DInput:a_bPhysicalDI[35] AT %IX."X20DI9372a".DigitalInput11;
	::DInput:a_bPhysicalDI[36] AT %IX."X20DI9372a".DigitalInput12;
	::DOutput:a_bPhysicalDO[19] AT %QX."X20DO9321-X8".DigitalOutput01;
	::DOutput:a_bPhysicalDO[20] AT %QX."X20DO9321-X8".DigitalOutput02;
	::DOutput:a_bPhysicalDO[21] AT %QX."X20DO9321-X8".DigitalOutput03;
	::DOutput:a_bPhysicalDO[22] AT %QX."X20DO9321-X8".DigitalOutput04;
	::DOutput:a_bPhysicalDO[23] AT %QX."X20DO9321-X8".DigitalOutput05;
	::DOutput:a_bPhysicalDO[24] AT %QX."X20DO9321-X8".DigitalOutput06;
	::DOutput:a_bPhysicalDO[25] AT %QX."X20DO9321-X8".DigitalOutput07;
	::DOutput:a_bPhysicalDO[26] AT %QX."X20DO9321-X8".DigitalOutput08;
	::DOutput:a_bPhysicalDO[27] AT %QX."X20DO9321-X8".DigitalOutput09;
	::DOutput:a_bPhysicalDO[28] AT %QX."X20DO9321-X8".DigitalOutput10;
	::DOutput:a_bPhysicalDO[29] AT %QX."X20DO9321-X8".DigitalOutput11;
	::DOutput:a_bPhysicalDO[30] AT %QX."X20DO9321-X8".DigitalOutput12;
END_VAR
```

## Logical view

Binary libraries used (declarations not repeated): standard, runtime, astime, asstring, operator, AsIecCon, AsCANopen, visapi, FileIO, AsIODiag, AsMem, dvframe, AsOpcUac, AsARCfg, sys_lib, AsTCP, AsIORTI, brsystem, AsFltGen, AsUSB, AsRfbExt 4.72.3, MpCom 1.65.1, MpBase 5.02.0, MpRecipe 1.65.1, Acp10man 3.18.2, Acp10par 3.18.2, NcGlobal 3.18.2, Acp10_MC 3.18.2, NtBuffer 5.00.6, NtMem 5.00.0, NtOvenInfo 5.00.0, NtRS232 5.00.2, NtStepper 5.00.0, NtFileIO 5.00.0, NtLogFile 5.00.1, NtTLBuz 5.00.2, NtMotion 5.00.9, NtPneu 5.00.0, NtConv 5.00.3, NtTCP 5.00.2, NtMessage 5.00.1, NtSMEMA 5.00.6, NtOPCUA 5.00.0, NtVersion 5.01.1, NtLF 5.01.5, NtRecipe 5.00.5
